		ClearWorkAreaLGVDone := TRUE;
		LGVAccessOK := FALSE;
		LGVCase := LGVCase + 1;	
		TFTimerSet(ADR(TimerOkBarriereSicurezze),5000, TRUE);	
		FOR iPost:=1 TO MAXAREAPRESENT DO
			IF LGV_Stato_Operazione^[k] = LGV_DEPOSITO_EFFETTUATO THEN  
				LGV_Stato_Operazione^[k] := LGV_OPERAZIONE_VERIFICATA;
				IF PH_WorkArea[k] THEN	//Se la fatocellula è ON
					IF TFMachinePalletizerMain.TEST_ENABLE THEN//Se sono in simulazione setto a TRUE la fotocellula virtuale
						I_PHPresenzaPalletVirtuale[k] := TRUE;
					ELSE
						//IF WorkArea^[k].Typology = TYPOLOGY_STACK OR WorkArea^[k].Typology = TYPOLOGY_LAYER THEN
						//	TFClearWorkAreaStack(WorkArea,WorkAreaState,k);
						//END_IF	
					END_IF
				ELSE 					//Se la fotocellula è OFF
					IF TFMachinePalletizerMain.TEST_ENABLE THEN//Se sono in simulazione setto a TRUE la fotocellula virtuale
						I_PHPresenzaPalletVirtuale[k] := TRUE;
					ELSE
						//IF WorkArea^[k].Typology = TYPOLOGY_STACK OR WorkArea^[k].Typology = TYPOLOGY_LAYER THEN
						//	TFClearWorkAreaStack(WorkArea,WorkAreaState,k);
						//END_IF	
						LGVErrorCode := ErrMACHINEPALLETIZER_PHOFFDOPODEPOSITO;
						LGVCase := 0;
					END_IF
				END_IF
			ELSIF LGV_Stato_Operazione^[k] = LGV_PRELIEVO_EFFETTUATO AND PH_WorkArea[k] THEN  
				LGV_Stato_Operazione^[k] := LGV_OPERAZIONE_VERIFICATA;
				IF NOT PH_WorkArea[k] THEN //Se la fotocellula è OFF
					IF TFMachinePalletizerMain.TEST_ENABLE THEN//Se sono in simulazione setto a FALSE la fotocellula virtuale
						I_PHPresenzaPalletVirtuale[k] := FALSE;
						TFClearWorkArea(WorkArea,WorkAreaState,k);
					ELSE
						TFClearWorkArea(WorkArea,WorkAreaState,k);
					END_IF
				ELSE					//Se la fotocellula è ON
					IF TFMachinePalletizerMain.TEST_ENABLE THEN//Se sono in simulazione setto a FALSE la fotocellula virtuale
						I_PHPresenzaPalletVirtuale[k] := FALSE;
						TFClearWorkArea(WorkArea,WorkAreaState,k);
					ELSE
						TFClearWorkArea(WorkArea,WorkAreaState,k);
					END_IF
					LGVErrorCode := ErrMACHINEPALLETIZER_PHONDOPOPRELIEVO;
					LGVCase := 0;
				END_IF
			ELSIF LGV_Stato_Operazione^[k] = LGV_OPERAZIONE_VERIFICATA THEN
				LGVErrorCode := ErrMACHINEPALLETIZER_MANCATOAGGIORNAMENTOSTATO;		
				LGVCase := 0;	
			END_IF
		END_FOR
			
	(* Case 7 - Power ON *)
	7:	
		IF BarriereSicurezzaEsterneOK THEN
			TFParametersArrayClear(ADR(ParametersArray));
			ParametersArray.Parameters[0] := '1';
			TFCommandSend(CmdPOWER,ParametersArray,MachineCmd^);
			LGV_ResetSW_RicIng := TRUE;
			LGVCase := LGVCase + 1;	
		ELSIF TFTimerDone(ADR(TimeoutControlloBarriereSicurezza)) THEN
			LGVErrorCode := ErrMACHINEPALLETIZER_BARRIEREOCCUPATE_LGVREQ_OFF;
			LGVCase := 0;
		END_IF	
			
	(* Case 8 - Power On OK *)
	8:	IF TFStateCodeGet(MachineState^) = StatePOWER_END OR
			TFIsModuleError(MachineError^) THEN
			LGV_ResetSW_RicIng := FALSE;
			LGVCase := LGVCase + 1;	
		END_IF
		
	(* Case 9 - Cmd DO *)
	9:	
		IF MachineWasRunning AND
			MachineMode^.Auto AND
			NOT MachineMode^.StopRequest AND
			NOT MachineMode^.RapidStopRequest AND NOT GateAccessActive THEN
			(*AND (SecurityGateStatus OR NOT ControlGateSecurity^*) 
			TFParametersArrayClear(ADR(ParametersArray));
			TFCommandSend(CmdDO,ParametersArray,MachineCmd^);
		END_IF
		LGVCase := 0;
	
	ELSE
		LGVAccessERROR := TRUE;
		LGVCase := 0;
	
END_CASE

(* Clocks *)
IF TFTimerDone(ADR(Timer100)) THEN
	TFTimerSet(ADR(Timer100),100,TRUE);
	Clock100 := NOT Clock100;
END_IF
IF TFTimerDone(ADR(Timer200)) THEN
	TFTimerSet(ADR(Timer200),200,TRUE);
	Clock200 := NOT Clock200;
END_IF
IF TFTimerDone(ADR(Timer1000)) THEN
	TFTimerSet(ADR(Timer1000),1000,TRUE);
	Clock1000 := NOT Clock1000;
END_IF

(* Se ho un errore durante la richiesta di ingresso, resetto esternamente gli HandShake *)
IF LGVErrorCode <> 0 THEN
	LGVResetHSKSUPNAV := TRUE;
END_IF


(* Access Lamp *)
LGVAccessLamp := ((LGVAccessOK AND Clock200) OR
				(LampadaIngressoInCorso AND Clock1000))AND
				NOT LGVAccessERROR OR (LGVAccessERROR AND Clock100);

END_FUNCTION_BLOCK

// ---- POUs/TFMachines/Utility/TFWorkflowsCheckState.TcPOU
FUNCTION TFWorkflowsCheckState : BOOL
VAR_INPUT
	WorkFlow : POINTER TO ARRAY[0..MAXWORKFLOW] OF WorkFlow;
	State : UINT; // stato da verificare
END_VAR
VAR
	i: UINT;
END_VAR
//Funzione che restituisce TRUE se tutti i WORFLOW sono nello stato richiesto

FOR i:=0 TO MAXWORKFLOW DO
	IF WorkFlow^[i].State <> State THEN
		RETURN;
	END_IF
END_FOR
TFWorkflowsCheckState := TRUE;

END_FUNCTION

// ---- POUs/TFModules/DataBase/TFSPRicavaDatiDaBarcodeUDC.TcPOU
FUNCTION_BLOCK TFSPRicavaDatiDaBarcodeUDC
VAR_INPUT
	BarcodeUDC 	: STRING;//Barcode in ingresso
	IDUDC 		: UDINT;//ID univoco che la macchina genera per ogni elemento depositato
	StartRead 	: BOOL;//Start lettura dati
	DBID		: UDINT;//ID del database, da ricavare dal configuratore
	AbilitaSTHere : BOOL;
	ResetError : bool;
END_VAR
VAR_OUTPUT
	DataFromDB 	: Record_From_DB; //Dati ricavati dal DB
	RecordID    : DINT; //se <> da 0 significa che l'elemento può entrare e rappresenta l'ordine di lavoro
	State 		: ARRAY [1..2] OF StoredProcedureState;
END_VAR
VAR
	nState: BYTE;
	arrParaList1: ARRAY [0..0] OF ST_DBParameter;
	arrParaList2: ARRAY [0..6] OF ST_DBParameter;
	SP_TryUdcCheckIn : FB_DBStoredProceduresRecordArray;
	SP_TryQtyCheckIn : FB_DBStoredProceduresRecordArray;

	bBusy: BOOL;
	bErr: BOOL;
	nErrid: UDINT;

	StateSP1 		: StoredProcedureState;
	StateSP2 		: StoredProcedureState;

	CalibroLocal : STRING;

END_VAR

CASE nState OF
	(*Idle*)
	0:
		IF StartRead THEN
			nState := 1;
			State[1].ReadRun := TRUE;
			DataFromDB.ArticleCode 	:= '';
			DataFromDB.Caliber		:= '';
			DataFromDB.Choice		:= '';
			DataFromDB.Length_mm	:= 0;
			DataFromDB.Quantity		:= 0;
			DataFromDB.Thickness_mm	:= 0;
			DataFromDB.Tone			:= '';
			DataFromDB.Udc			:= '';
			DataFromDB.Width_mm		:= 0;
		END_IF
	(* Case 1 : Init Dei parametri per esecuzione SP *)
	1:
		arrParaList1[0].sParameterName 		:= '@Udc';
		arrParaList1[0].eParameterDataType 	:= eDBColumn_NVarChar;
		arrParaList1[0].eParameterType 		:= eDBParameter_Input;
		arrParaList1[0].cbParameterValue 	:= SIZEOF(BarcodeUDC);
		arrParaList1[0].pParameterValue 		:= ADR(BarcodeUDC);
		SP_TryUdcCheckIn.bExecute := TRUE;
		
		(*SP_TryUdcCheckIn(
				sNetID	:= ,
				hDBID	:= DBID,
				sProcedureName	:= 'TryUdcCheckIn',
				cbParameterList	:= SIZEOF(arrParaList1),
				pParameterList	:= ADR(arrParaList1),
				nStartIndex		:= 0,
				nRecordCount	:= 1,
				cbRecordArraySize	:= SIZEOF(DataFromDB),
				pDestAddr			:= ADR(DataFromDB),
				//bExecute			:= TRUE,
				tTimeout			:= T#50S,
				bBusy				=> bBusy,
				bError				=> State[1].Error,
				nErrID				=> State[1].ErrorID,
				sSQLState			=> State[1].Sqlstate,
				nRecords			=> State[1].NumeroRecordLetti);	*)
		//IF NOT SP_TryUdcCheckIn.bBusy THEN
			nState := 2;
		//	SP_TryUdcCheckIn.bExecute := FALSE;
		//END_IF

	(*Start stored procedure "TryUdcCheckIn"*)
	2:
		IF NOT SP_TryUdcCheckIn.bBusy THEN
			SP_TryUdcCheckIn.bExecute := FALSE;
			IF AbilitaSTHere THEN
				nState := 10;
				RecordID := 0;
			ELSE
				nState := 12;
				State[2].ReadRun 	:= FALSE;
				State[2].ReadDone 	:= TRUE;
			END_IF
			State[1].ReadRun 	:= FALSE;
			State[1].ReadDone 	:= TRUE;
		END_IF
	
	10:
		//Parametro UDC generato dalla linea di ingresso
		arrParaList2[0].sParameterName 		:= '@IdEnteringUnit';
		arrParaList2[0].eParameterDataType 	:= eDBColumn_BigInt;
		arrParaList2[0].eParameterType 		:= eDBParameter_Input;
		arrParaList2[0].cbParameterValue 	:= SIZEOF(IDUDC);
		arrParaList2[0].pParameterValue 		:= ADR(IDUDC);

		//Parametro BARCODE
		arrParaList2[1].sParameterName 		:= '@UDC';
		arrParaList2[1].eParameterDataType 	:= eDBColumn_NVarChar;
		arrParaList2[1].eParameterType 		:= eDBParameter_Input;
		arrParaList2[1].cbParameterValue 	:= SIZEOF(BarcodeUDC);
		arrParaList2[1].pParameterValue 	:= ADR(BarcodeUDC);
		
		//Parametro Articolo
		arrParaList2[2].sParameterName 		:= '@Articolo';
		arrParaList2[2].eParameterDataType 	:= eDBColumn_NVarChar;
		arrParaList2[2].eParameterType 		:= eDBParameter_Input;
		arrParaList2[2].cbParameterValue 	:= SIZEOF(DataFromDB.ArticleCode);
		arrParaList2[2].pParameterValue 		:= ADR(DataFromDB.ArticleCode);
		//Parametro Scelta
		arrParaList2[3].sParameterName 		:= '@Scelta';
		arrParaList2[3].eParameterDataType 	:= eDBColumn_NVarChar;
		arrParaList2[3].eParameterType 		:= eDBParameter_Input;
		arrParaList2[3].cbParameterValue 	:= SIZEOF(DataFromDB.Choice);
		arrParaList2[3].pParameterValue 		:= ADR(DataFromDB.Choice);

		//Parametro tono
		arrParaList2[4].sParameterName 		:= '@Tono';
		arrParaList2[4].eParameterDataType 	:= eDBColumn_NVarChar;
		arrParaList2[4].eParameterType 		:= eDBParameter_Input;
		arrParaList2[4].cbParameterValue 	:= SIZEOF(DataFromDB.Tone);
		arrParaList2[4].pParameterValue 		:= ADR(DataFromDB.Tone);

		//Parametro Calibro
		arrParaList2[5].sParameterName 		:= '@Calibro';
		arrParaList2[5].eParameterDataType 	:= eDBColumn_NVarChar;
		arrParaList2[5].eParameterType 		:= eDBParameter_Input;

		arrParaList2[5].cbParameterValue 	:= SIZEOF(DataFromDB.Caliber);
		arrParaList2[5].pParameterValue 		:= ADR(DataFromDB.Caliber);
		//Parametro Quantità
		arrParaList2[6].sParameterName 		:= '@Quantity';
		arrParaList2[6].eParameterDataType 	:= eDBColumn_Float;
		arrParaList2[6].eParameterType 		:= eDBParameter_Input;
		arrParaList2[6].cbParameterValue 	:= SIZEOF(DataFromDB.Quantity);
		arrParaList2[6].pParameterValue 	:= ADR(DataFromDB.Quantity);
		//Reset variabile risultante
		//RecordID := 0;
		//Lancio Comando
		SP_TryQtyCheckIn.bExecute := TRUE;

		(*SP_TryQtyCheckIn(
				sNetID	:= ,
				hDBID	:= DBID,
				sProcedureName	:= 'TryQtyCheckIn',
				cbParameterList	:= SIZEOF(arrParaList2),
				pParameterList	:= ADR(arrParaList2),
				nStartIndex		:= 0,
				nRecordCount	:= 1,
				cbRecordArraySize	:= SIZEOF(RecordID),
				pDestAddr			:= ADR(RecordID),
				//bExecute			:= TRUE,
				tTimeout			:= T#50S,
				bBusy				=> bBusy,
				bError				=> State[2].Error,
				nErrID				=> State[2].ErrorID,
				sSQLState			=> State[2].Sqlstate,
				nRecords			=> State[2].NumeroRecordLetti);*)
		
		State[2].ReadRun 	:= TRUE;
		State[2].ReadDone 	:= FALSE;

		//IF NOT SP_TryQtyCheckIn.bBusy THEN
		//	SP_TryQtyCheckIn.bExecute := FALSE;
			nState := 11;
		//END_IF

	(*Start stored procedure "TryUdcCheckIn"*)
	11:
		IF NOT SP_TryQtyCheckIn.bBusy THEN
			SP_TryQtyCheckIn.bExecute := FALSE;
			nState := 12;//3;
			State[2].ReadRun 	:= FALSE;
			State[2].ReadDone 	:= TRUE;
		END_IF

	(* Attesa che il comando dall'esterno venga azzerato *)	
	12:
		IF NOT StartRead OR ResetError THEN 
			nState := 0;
			State[1].ReadRun 	:= FALSE;
			State[2].ReadRun 	:= FALSE;
			State[1].ReadDone 	:= FALSE;
			State[2].ReadDone 	:= FALSE;
			SP_TryUdcCheckIn.bExecute := FALSE;
			SP_TryQtyCheckIn.bExecute := FALSE;
			
		END_IF	
		
END_CASE

//Lancio SP
(*
IF ResetError THEN
	IF SP_TryUdcCheckIn.bError AND NOT SP_TryUdcCheckIn.bBusy THEN
		SP_TryUdcCheckIn.bExecute := FALSE;
		//SP_TryUdcCheckIn(bExecute := FALSE);
	END_IF
	IF  SP_TryQtyCheckIn.bError AND NOT SP_TryUdcCheckIn.bBusy THEN 
		SP_TryQtyCheckIn.bExecute := FALSE;
		//SP_TryQtyCheckIn(bExecute := FALSE);
	END_IF
	ResetError := FALSE;
END_IF
*)

SP_TryUdcCheckIn(
				sNetID	:= ,
				hDBID	:= DBID,
				sProcedureName	:= 'TryUdcCheckIn',
				cbParameterList	:= SIZEOF(arrParaList1),
				pParameterList	:= ADR(arrParaList1),
				nStartIndex		:= 0,
				nRecordCount	:= 1,
				cbRecordArraySize	:= SIZEOF(DataFromDB),
				pDestAddr			:= ADR(DataFromDB),
				//bExecute			:= TRUE,
				tTimeout			:= T#50S,
				bBusy				=> bBusy,
				bError				=> State[1].Error,
				nErrID				=> State[1].ErrorID,
				sSQLState			=> State[1].Sqlstate,
				nRecords			=> State[1].NumeroRecordLetti);

//Lancio SP
SP_TryQtyCheckIn(
				sNetID	:= ,
				hDBID	:= DBID,
				sProcedureName	:= 'TryQtyCheckIn',
				cbParameterList	:= SIZEOF(arrParaList2),
				pParameterList	:= ADR(arrParaList2),
				nStartIndex		:= 0,
				nRecordCount	:= 1,
				cbRecordArraySize	:= SIZEOF(RecordID),
				pDestAddr			:= ADR(RecordID),
				//bExecute			:= TRUE,
				tTimeout			:= T#50S,
				bBusy				=> bBusy,
				bError				=> State[2].Error,
				nErrID				=> State[2].ErrorID,
				sSQLState			=> State[2].Sqlstate,
				nRecords			=> State[2].NumeroRecordLetti);

//reset errori SP				
IF ResetError THEN
	IF State[1].Error THEN
		State[1].Error := FALSE;
	END_IF
	IF State[2].Error THEN 
		State[2].Error := FALSE;
	END_IF
	ResetError := FALSE;
END_IF

END_FUNCTION_BLOCK

// ---- POUs/TFModules/DataBase/TFSPRichiestaIngressoMateriale.TcPOU
FUNCTION_BLOCK TFSPRichiestaIngressoMateriale
VAR_INPUT
	BarcodeUDC 	: STRING;//Barcode in ingresso
	StartRead 	: BOOL;//Start lettura dati
	DBID		: UDINT;//ID del database, da ricavare dal configuratore
END_VAR
VAR_OUTPUT
	DataFromDB 	: Record_From_DB; //Dati ricavati dal DB
	State 		: StoredProcedureState;
END_VAR
VAR
	nState: BYTE;
	arrParaList: ARRAY [0..0] OF ST_DBParameter;
	SP_RecordArray : FB_DBStoredProceduresRecordArray;
	bBusy: BOOL;
	bErr: BOOL;
	nErrid: UDINT;
	DataFromDB1 	: Record_From_DB; //Dati ricavati dal DB
END_VAR

CASE nState OF
	(*Idle*)
	0:
		IF StartRead THEN
			nState := 1;
			State.ReadRun := TRUE;
		END_IF
	(* Case 1 : Init Dei parametri per esecuzione SP *)
	1:
		arrParaList[0].sParameterName 		:= '@Udc';
		arrParaList[0].eParameterDataType 	:= eDBColumn_NVarChar;
		arrParaList[0].eParameterType 		:= eDBParameter_Input;
		arrParaList[0].cbParameterValue 	:= SIZEOF(BarcodeUDC);
		arrParaList[0].pParameterValue 		:= ADR(BarcodeUDC);
	
		DataFromDB.ArticleCode 	:= '';
		DataFromDB.Caliber		:= '';
		DataFromDB.Choice		:= '';
		DataFromDB.Length_mm	:= 0;
		DataFromDB.Quantity		:= 0;
		DataFromDB.Thickness_mm	:= 0;
		DataFromDB.Tone			:= '';
		DataFromDB.Udc			:= '';
		DataFromDB.Width_mm		:= 0;

		SP_RecordArray.bExecute := TRUE;
		
		nState := 2;

	(*Start stored procedure "TryUdcCheckIn"*)
	2:
		
		
		IF NOT SP_RecordArray.bBusy THEN
			SP_RecordArray.bExecute := FALSE;
			nState := 3;
			State.ReadRun 	:= FALSE;
			State.ReadDone 	:= TRUE;
		END_IF
	
	(* Attesa che il comando dall'esterno venga azzerato *)	
	3:
		IF NOT StartRead THEN 
			nState := 0;
			State.ReadRun 	:= FALSE;
			State.ReadDone 	:= FALSE;
		END_IF	
		
END_CASE

//Lancio FB
SP_RecordArray(
				sNetID	:= ,
				hDBID	:= DBID,
				sProcedureName	:= 'TryUdcCheckIn',
				cbParameterList	:= SIZEOF(arrParaList),
				pParameterList	:= ADR(arrParaList),
				nStartIndex		:= 0,
				nRecordCount	:= 1,
				cbRecordArraySize	:= SIZEOF(DataFromDB1),
				pDestAddr			:= ADR(DataFromDB1),
				//bExecute			:= TRUE,
				tTimeout			:= T#50S,
				bBusy				=> bBusy,
				bError				=> State.Error,
				nErrID				=> State.ErrorID,
				sSQLState			=> State.Sqlstate,
				nRecords			=> State.NumeroRecordLetti);

END_FUNCTION_BLOCK

// ---- POUs/TFModules/DataBase/TFVerificaLetturaBarcodeConDatiDB.TcPOU
FUNCTION_BLOCK TFVerificaLetturaBarcodeConDatiDB //FB che verifica se i dati letti del barcode sono validi per il database
VAR_INPUT
	VerificaDati 	: BOOL;	//Bit di start
	BarcodeUDC 		: STRING;//Barcode elemento
	IDUDC 			: UDINT;//ID elemento
	AbilitaSTHere 	: BOOL;
END_VAR
VAR
	DataElementNull : TFMachinePalletizer_DataElement;
	DimElementNull	: TFDimensionElement; 
	RicavaDatiDaBarcodeUDC : TFSPRicavaDatiDaBarcodeUDC;
	FirstCycleDone : bool;
END_VAR
VAR_OUTPUT
	DatoValido 			: BOOL; //Dati ok
	VerificaDatiDone 	: BOOL; //Verifica completata
	DataElement 		: TFMachinePalletizer_DataElement;//dati elemento
	DimElement 			: TFDimensionElement; //Dimensioni Pezzi
	RequetsIDValido		: BOOL;//se TRUE allora il materiale puù entrare
	Error : BOOL;
END_VAR


IF VerificaDati AND BarcodeUDC <> '0' AND BarcodeUDC <> '' AND NOT (RicavaDatiDaBarcodeUDC.State[1].Error OR RicavaDatiDaBarcodeUDC.State[2].Error) THEN//Se ho il comando di verifica dei dati su DB
	Error 			:= FALSE;
	RicavaDatiDaBarcodeUDC.ResetError := FALSE;
	RequetsIDValido := FALSE;
	DataElement 	:= DataElementNull;
	DimElement 		:= DimElementNull;
	AbilitaSTHere 	:= TRUE;	

	(* Eseguo Stored Procedure per acquisire i dati dell'articolo all'interno dell'UDC avente il codice in ingresso del BARCODE *)
	RicavaDatiDaBarcodeUDC.BarcodeUDC 	:= BarcodeUDC; 	//BARCODE letto sull'elemento
	RicavaDatiDaBarcodeUDC.DBID 		:= 1;			//Numero del DB configurato
	RicavaDatiDaBarcodeUDC.IDUDC 		:= IDUDC;		//ID dell'elemento
	RicavaDatiDaBarcodeUDC.StartRead 	:= TRUE;		//Start comando lettura
	RicavaDatiDaBarcodeUDC.AbilitaSTHere := AbilitaSTHere;	

	IF (RicavaDatiDaBarcodeUDC.State[1].ReadDone AND NOT RicavaDatiDaBarcodeUDC.State[1].Error) THEN
		//Dati elemento
		DataElement.Tono 	:= RicavaDatiDaBarcodeUDC.DataFromDB.Tone;
		DataElement.Scelta 	:= RicavaDatiDaBarcodeUDC.DataFromDB.Choice;
		DataElement.Calibro := RicavaDatiDaBarcodeUDC.DataFromDB.Caliber;
		DataElement.Codice  := RicavaDatiDaBarcodeUDC.DataFromDB.ArticleCode;
		DataElement.Quantity := LREAL_TO_UINT(RicavaDatiDaBarcodeUDC.DataFromDB.Quantity);
		DataElement.ArticleDescription  := RicavaDatiDaBarcodeUDC.DataFromDB.ArticleDescription;
		
		//Dimensioni elemento
		DimElement.ZDim		:= DINT_TO_REAL(RicavaDatiDaBarcodeUDC.DataFromDB.Thickness_mm);
		IF RicavaDatiDaBarcodeUDC.DataFromDB.Length_mm > RicavaDatiDaBarcodeUDC.DataFromDB.Width_mm THEN
			DimElement.XDim		:= DINT_TO_REAL(RicavaDatiDaBarcodeUDC.DataFromDB.Length_mm);
			DimElement.YDim		:= DINT_TO_REAL(RicavaDatiDaBarcodeUDC.DataFromDB.Width_mm);
		ELSE
			DimElement.XDim		:= DINT_TO_REAL(RicavaDatiDaBarcodeUDC.DataFromDB.Width_mm);
			DimElement.YDim		:= DINT_TO_REAL(RicavaDatiDaBarcodeUDC.DataFromDB.Length_mm);
		END_IF

		//Validità dati
		DatoValido 			:= NOT RicavaDatiDaBarcodeUDC.State[1].Error AND DataElement.Codice <> '0' AND DataElement.Codice <> '';
		 
		IF ((RicavaDatiDaBarcodeUDC.State[2].ReadDone AND NOT RicavaDatiDaBarcodeUDC.State[2].Error) OR NOT AbilitaSTHere) THEN//Se lettura da DB terminata	
			//Valore Record ID che se <> da 0 vuol dire che il materiale puù entrare
			IF NOT RicavaDatiDaBarcodeUDC.State[2].Error THEN
				DataElement.WorkingID 	:= DINT_TO_STRING(RicavaDatiDaBarcodeUDC.RecordID);
				RequetsIDValido 		:= DataElement.WorkingID <> '0';//indico che l'elemento può entrare
				IF NOT RequetsIDValido THEN
					DataElement.WorkingID := '0';
				END_IF
			ELSE
				DataElement.WorkingID 	:= '';
			END_IF
		END_IF
		RicavaDatiDaBarcodeUDC.StartRead := FALSE;//Stoppo la lettura
		VerificaDatiDone 	:= TRUE;
	ELSIF FirstCycleDone AND RicavaDatiDaBarcodeUDC.State[1].Error OR RicavaDatiDaBarcodeUDC.State[2].Error THEN
		Error 				:= TRUE;
		VerificaDatiDone 	:= TRUE;
		RicavaDatiDaBarcodeUDC.StartRead := FALSE;//Stoppo la lettura
	END_IF
	FirstCycleDone := TRUE;
	
ELSIF VerificaDatiDone AND NOT VerificaDati THEN //Attendo che dall'esterno venga terminata la richiesta di lettura dal DB
	DatoValido 			:= FALSE;
	VerificaDatiDone 	:= FALSE;
	FirstCycleDone 		:= FALSE;
ELSIF RicavaDatiDaBarcodeUDC.State[1].Error OR RicavaDatiDaBarcodeUDC.State[2].Error THEN
	DatoValido 	:= FALSE;
	RicavaDatiDaBarcodeUDC.ResetError := TRUE;
	Error 				:= TRUE;
END_IF

//Esguo FB per ricerca dati da DB
RicavaDatiDaBarcodeUDC();

END_FUNCTION_BLOCK

// ---- POUs/TFModules/Misurazione Ingresso/TFGestioneFTC_Misura.TcPOU
FUNCTION_BLOCK TFGestioneFTC_Misura
VAR_INPUT
	EseguiMisura 	: BOOL; //Start esecuzione misura
	IN 				: TFGestioneFTC_Misura_IN; //Struttura Ingressi
	PosizioneAsse 	: LREAL;	//Posizione dell'asse
	AsseInMovimento : BOOL; //Indica se l'asse è in movimento o meno
	SpazioFiltro 	: REAL := 50; //Spazio utilizzato per filtrare le FTC
END_VAR
VAR_OUTPUT
	
	OUT 				: TFGestioneFTC_Misura_OUT;
END_VAR
VAR
	FiltroFTC1 : Signal_SpaceFilter;
	FiltroFTC2 : Signal_SpaceFilter;
	FiltroFTC3 : Signal_SpaceFilter;
	FiltroFTC4 : Signal_SpaceFilter;
	
	StartLettura 	: BOOL;
	PosizioneTesta 	: REAL;
	PosizioneCoda 	: REAL;
	
	UltimaLunghezza : REAL := 0; //Appoggio x debug
	FTC_PallettoneIntercettata : BOOL;
END_VAR

FiltroFTC1(Sensor:=IN.FTC_ZoccoloBasso,
			ActualPosition:=PosizioneAsse,
			SpaceFilter:=SpazioFiltro,
			AxisMoving:=AsseInMovimento,
			EnableDirectStatusAxStop:=TRUE,
			SensorOUT=>OUT.FTC_ZoccoloBassoFiltrata);
FiltroFTC2(Sensor:=IN.FTC_Pallettone,
			ActualPosition:=PosizioneAsse,
			SpaceFilter:=SpazioFiltro,
			AxisMoving:=AsseInMovimento,
			EnableDirectStatusAxStop:=TRUE,
			SensorOUT=>OUT.FTC_PallettoneFiltrata);
FiltroFTC3(Sensor:=IN.FTC_CavallinaBassa,
			ActualPosition:=PosizioneAsse,
			SpaceFilter:=SpazioFiltro,
			AxisMoving:=AsseInMovimento,
			EnableDirectStatusAxStop:=TRUE,
			SensorOUT=>OUT.FTC_CavallinaBassaFiltrata);
FiltroFTC4(Sensor:=IN.FTC_CavallinaAlta,
			ActualPosition:=PosizioneAsse,
			SpaceFilter:=SpazioFiltro,
			AxisMoving:=AsseInMovimento,
			EnableDirectStatusAxStop:=TRUE,
			SensorOUT=>OUT.FTC_CavallinaAltaFiltrata);

IF EseguiMisura THEN
	IF OUT.FTC_ZoccoloBassoFiltrata THEN
		//Memorizzo la quota della testa dell'elemento
		IF NOT StartLettura THEN 
			Out.Supporto := SupportoVuoto;//Sbianco la memoria dell'ultima lettura
			UltimaLunghezza := 0;
			OUT.MisuraInCorso := TRUE;  
			PosizioneTesta := PosizioneAsse;
			StartLettura := TRUE;
		END_IF	
	
		IF OUT.FTC_PallettoneFiltrata OR WEINTEK_TRANSPORT.AbilitaIngressoPalletSingolo THEN //Se vedo questa FTC sicuramente non è una cassa
			IF NOT WEINTEK_TRANSPORT.AbilitaIngressoPalletSingolo THEN
				OUT.Supporto.Tipologia := PALLET_ACCOPPIATI;//Dichiaro la tipologia di supporto
			ELSE
				OUT.Supporto.Tipologia := PALLET_STANDARD;//Dichiaro la tipologia di supporto
			END_IF
			OUT.Supporto.ZDim := 1000;//800;
			OUT.Supporto.HMAX := 1000;//800;
			FTC_PallettoneIntercettata := TRUE;
			IF OUT.FTC_CavallinaBassaFiltrata THEN //Se vedo questa FTC si tratta di una cavallina Bassa
				OUT.Supporto.Tipologia := CAVALLETTO;//Dichiaro la tipologia di supporto
				OUT.Supporto.ZDim := 350;
				OUT.Supporto.HMAX := 1600;
			END_IF
			IF OUT.FTC_CavallinaAltaFiltrata THEN //Se vedo questa FTC si tratta di cavallina ALTA
				OUT.Supporto.Tipologia := CAVALLETTO;//Dichiaro la tipologia di supporto
				OUT.Supporto.ZDim := 350;
				OUT.Supporto.HMAX := 2000;
			END_IF
		ELSIF NOT OUT.FTC_PallettoneFiltrata AND NOT FTC_PallettoneIntercettata THEN //Se non vedo questa FTC si tratta di una cassa
			OUT.Supporto.Tipologia := CASSA_STANDARD;//Dichiaro la tipologia di supporto
			OUT.Supporto.ZDim := 200;
			OUT.Supporto.HMAX := 420;
		END_IF
	
	ELSIF NOT OUT.FTC_ZoccoloBassoFiltrata AND StartLettura THEN
		Out.MisuraDone := TRUE;
		OUT.MisuraInCorso := TRUE;  
		PosizioneCoda := PosizioneAsse;
		Out.LunghezzaMisurata := PosizioneCoda - PosizioneTesta;
		Out.Supporto.XDim := Out.LunghezzaMisurata;
		UltimaLunghezza := Out.LunghezzaMisurata;
		FTC_PallettoneIntercettata := FALSE;
	END_IF
	//Cambio tipologia nel caso di pallet >= 1400
	IF Out.Supporto.XDim >= 1400 AND OUT.Supporto.Tipologia = PALLET_ACCOPPIATI THEN
		OUT.Supporto.Tipologia := PALLET_STANDARD;
	END_IF
ELSE
	Out.MisuraDone 		:= FALSE;
	OUT.MisuraInCorso 	:= FALSE;
	StartLettura 		:= FALSE;
	
END_IF

END_FUNCTION_BLOCK

// ---- POUs/TFModules/Moduli TF/TFModulePalletizer_Pinza_mag.TcPOU
FUNCTION_BLOCK TFModulePalletizer_Pinza_mag
VAR_INPUT
	Cmd 	: CommandBuffer;
	Cfg 	: Config;
	IN 		: TFMchinePalletizer_PinzaVentose_IN;
	IN_Ax 	: Module_Palletizer_Ax_IN;
	
	AspirazioneDX1 : POINTER TO TF_VacumOVEM;
	AspirazioneSX1 : POINTER TO TF_VacumOVEM;
	AspirazioneDX2 : POINTER TO TF_VacumOVEM;
	AspirazioneSX2 : POINTER TO TF_VacumOVEM;

	CilindroSbloccoRotazione 	: POINTER TO SC_Cylinder;
	CilindroSbloccoBascolante 	: POINTER TO SC_Cylinder;
	CilindroApertura 			: POINTER TO DC_Cylinder;
	
	ModuleJ : POINTER TO TFModulePalletizer_Ax;
	ModuleK : POINTER TO TFModulePalletizer_Ax;

	ManCmd 				: POINTER TO TFMachinePalletizer_PinzaVentoseManCmd;
	ElementoInPrelievo 	: TFMachinePalletizer_PlaceElement;
	DataElement			: TFMachinePalletizer_DataElement; (* Struttura dati che la macchina acquisisce/trasferisce in fase di pallettizzazione/depallettizazione *)
	PrelievoSuMagazino : BOOL;//indica che il prelievo è su cavallina

	Mission : POINTER TO TFMachinePalletizer_Mission;
	AbilitazioneSbloccoRotazione 	: BOOL;//Abilitazione sblocco rotazione pinza
	AbilitazioneSbloccoBascolante 	: BOOL;//Abilitazione sblocco bascolante pinza	
	IN_SimulazioneSenzaHW : BOOL;
	AbilitaAperturaAutomaticaPinza : BOOL;//Abilitazione apertura automatica pinza
END_VAR
VAR_OUTPUT
	CmdExe 		: CommandExe;
	CmdExd 		: CommandExe;
	CmdNext 	: Command;
	CmdLog 		: CommandLog;
	ProgramLog 	: ProgrammaLog; 
	State 		: State;
	StateLog 	: StateLog;
	Error 		: Error;
	ErrorLog 	: ErrorLog;
	Warning 	: Warning;
	WarningLog	: WarningLog;
	OUT 		: TFMachinePalletizer_PinzaVentose_OUT;
	StatoPinza 	: TFMachinePalletizer_PinzaState;

END_VAR
VAR
	Power 	: UINT;
	Init 	: BOOL;
	Timer 	: REAL;
	Timeout : REAL;
	TimerAspirazione 	: REAL;
	ParametersArray 	: ParametersArray;
	MAN_Actuator 		: UINT;
	MAN_Cmd 			: UINT;

	DistanzaFTC_J0 		: REAL;
	DistanzaFTC_J180 	: REAL;
	DistanzaFTC_K0 		: REAL;
	DistanzaFTC_K180 	: REAL;

	TimerPresaPiastrella : REAL;		
	DisattivazioneTotaleAspirazioni : bool;
	ByPassAttesaDistacco : BOOL;

	DistanzaJForzata : REAL;
	DistanzaKForzata : REAL;

END_VAR

IF NOT Init THEN
	TFCommandBufferClear(ADR(Cmd));
	TFCommandClear(ADR(CmdNext));
	TFCommandExeClear(ADR(CmdExe));
	TFStateUpdate(ADR(State),StateNOP);
	TFErrorClear(ADR(Error));
	TFWarningClear(ADR(Warning));
	Init := TRUE;
END_IF

(* Generic Timer - Add here all your Timers *)
TFTimerCall(ADR(Timer),Cfg.TimeBase);
TFTimerCall(ADR(Timeout),Cfg.TimeBase);
TFTimerCall(ADR(TimerPresaPiastrella),Cfg.TimeBase);
TFTimerCall(ADR(TimerAspirazione),Cfg.TimeBase);
(* External To Buffered Command *)
TFCommandToNext(ADR(Cmd),ADR(CmdNext),ADR(CmdExe),ADR(Cfg),ADR(Error),ADR(ErrorLog),ADR(State));

(* Buffered To Exe Command *)
TFCommandToExecution(ADR(CmdNext),ADR(CmdExe),ADR(Error),ADR(ErrorLog),ADR(State),ADR(CmdLog));

(* Chiamata FB *)
AspirazioneDX1^();
AspirazioneSX1^();
AspirazioneDX2^();
AspirazioneSX2^();
CilindroSbloccoRotazione^();
CilindroSbloccoBascolante^();

DistanzaFTC_J0 		:= Keyence_LRTB2000C(IN.InKeyence_J0_Byte0,IN.InKeyence_J0_Byte1);
DistanzaFTC_J180	:= Keyence_LRTB2000C(IN.InKeyence_J180_Byte0,IN.InKeyence_J180_Byte1);
DistanzaFTC_K0 		:= Keyence_LRTB2000C(IN.InKeyence_K0_Byte0,IN.InKeyence_K0_Byte1);
DistanzaFTC_K180	:= Keyence_LRTB2000C(IN.InKeyence_K180_Byte0,IN.InKeyence_K180_Byte1);

OUT.DistanzaFTC_J0 		:= DistanzaFTC_J0; 		
OUT.DistanzaFTC_J180	:= DistanzaFTC_J180;	
OUT.DistanzaFTC_K0 		:= DistanzaFTC_K0; 		
OUT.DistanzaFTC_K180   	:= DistanzaFTC_K180; 

DistanzaJForzata:=0;
IF ABS(DistanzaFTC_J0-DistanzaFTC_J180) > 30 THEN
	DistanzaJForzata := MIN(DistanzaFTC_J0,DistanzaFTC_J180);
END_IF
DistanzaKForzata:=0;
IF ABS(DistanzaFTC_K0-DistanzaFTC_K180) > 30 THEN
	DistanzaKForzata := MIN(DistanzaFTC_K0,DistanzaFTC_K180);
END_IF
OUT.DistanzaMedia := (DistanzaFTC_J0 + 	
                 DistanzaFTC_J180 +
                 DistanzaFTC_K0 + 	
                 DistanzaFTC_K180)/4;
				 
IF DistanzaKForzata > 0 THEN
	OUT.DistanzaMedia := (DistanzaJForzata +
                 DistanzaFTC_K0 + 	
                 DistanzaFTC_K180)/3;
END_IF
IF DistanzaJForzata > 0 THEN
	OUT.DistanzaMedia := (DistanzaFTC_J0 + 	
                 DistanzaFTC_J180 +
                 DistanzaKForzata)/3;
END_IF
IF DistanzaKForzata > 0 AND DistanzaJForzata > 0 THEN
	OUT.DistanzaMedia := (DistanzaJForzata +
                 DistanzaKForzata)/2;
END_IF

(* Exe Command *)
CASE CmdExe.Code OF

	(* ******************************************************************************************************** *)
	(* Nop  *)
	(* ******************************************************************************************************** *)
	CmdNOP:	;			
	(* ******************************************************************************************************** *)
	(* Stop *)
	(* ******************************************************************************************************** *)
	CmdSTOP:
		CASE CmdExe.CmdCase OF
			
			(* Case 0 *)
			0: 	TFStateUpdate(ADR(State),StateSTOP_RUN);
				TFTimerSet(ADR(Timeout),500,TRUE);
				TFCommandCase(ADR(CmdExe),1,CommandCase_INC);

			(* Case 1 - Clear All Commands*)
			1:	
				TFCommandCase(ADR(CmdExe),100,CommandCase_JMP);
			(* Case 100 *)
			100:TFStateUpdate(ADR(State),StateSTOP_END);
				TFCommandExeClear(ADR(CmdExe));

			ELSE
				TFError(ErrNOCMDCASE,ErrNULL,ADR(CmdExe),ADR(State),ADR(Error),ADR(ErrorLog));
		END_CASE;
	
	(* ******************************************************************************************************** *)
	(* Error Reset *)
	(* ******************************************************************************************************** *)
	CmdRESET:
		CASE CmdExe.CmdCase OF

			(* Case 0 *)
			0: 	TFStateUpdate(ADR(State),StateRESET_RUN);
				TFTimerSet(ADR(Timeout),2000+100,TRUE);
				TFTimerSet(ADR(Timer),2000,TRUE);
				TFCommandCase(ADR(CmdExe),1,CommandCase_JMP);

			
			(* Case 1 - RESET COMANDI*)
			1: 
				TFClearAllCmdModulePinzaMagazzino(AspirazioneDX1,AspirazioneSX1,AspirazioneDX2,AspirazioneSX2,CilindroSbloccoRotazione,CilindroSbloccoBascolante);
				TFCommandCase(ADR(CmdExe),1,CommandCase_INC);
			
			(* Case 2 - Invio comando di reset *)
			2:
				AspirazioneDX1^.Command^.ErrorReset 				:= TRUE;	
				AspirazioneSX1^.Command^.ErrorReset 				:= TRUE;	
				AspirazioneDX2^.Command^.ErrorReset 				:= TRUE;	
				AspirazioneSX2^.Command^.ErrorReset 				:= TRUE;	
				CilindroSbloccoRotazione^.Command.ErrorReset 	:= TRUE;	
				CilindroSbloccoBascolante^.Command.ErrorReset 	:= TRUE;	
				TFCommandCase(ADR(CmdExe),1,CommandCase_INC);
			
			(* Case 3 - Invio comando di reset *)
			3:
				IF (AspirazioneDX1^.Status.ErrorResetDone AND AspirazioneDX2^.Status.ErrorResetDone AND
					AspirazioneSX1^.Status.ErrorResetDone AND AspirazioneSX2^.Status.ErrorResetDone AND
					CilindroSbloccoRotazione^.Status.ErrorResetDone AND CilindroSbloccoBascolante^.Status.ErrorResetDone) OR IN_SimulazioneSenzaHW THEN					
					TFClearAllCmdModulePinzaMagazzino(AspirazioneDX1,AspirazioneSX1,AspirazioneDX2,AspirazioneSX2,CilindroSbloccoRotazione,CilindroSbloccoBascolante);
					TFCommandCase(ADR(CmdExe),99,CommandCase_JMP);
				ELSIF TFTimerDone(ADR(Timer)) THEN
					TFClearAllCmdModulePinzaMagazzino(AspirazioneDX1,AspirazioneSX1,AspirazioneDX2,AspirazioneSX2,CilindroSbloccoRotazione,CilindroSbloccoBascolante);
					TFError(ErrTORESET,ErrNULL,ADR(CmdExe),ADR(State),ADR(Error),ADR(ErrorLog));
				END_IF

			(* Case 99 *)
			99:	TFErrorClear(ADR(Error));
				TFWarningClear(ADR(Warning));
				TFCommandCase(ADR(CmdExe),100,CommandCase_JMP);

			(* Case 100 *)
			100:TFStateUpdate(ADR(State),StateRESET_END);
				TFCommandExeClear(ADR(CmdExe));

			ELSE
				TFError(ErrNOCMDCASE,ErrNULL,ADR(CmdExe),ADR(State),ADR(Error),ADR(ErrorLog));
		END_CASE;

		(*IF AspirazioneDX^.Status.ErrorID <> ErrNULL THEN
			TFClearAllCmdModulePinza(AspirazioneDX,AspirazioneSX,CilindroApertura,CilindroSbloccoRotazione,AspirazioneFaldaDX,AspirazioneFaldaSX,CilindroTasteggio);
			TFError(ErrCYLINDER,AspirazioneDX^.Status.ErrorID,ADR(CmdExe),ADR(State),ADR(Error),ADR(ErrorLog));
		ELSIF AspirazioneSX^.Status.ErrorID <> ErrNULL THEN
			TFClearAllCmdModulePinza(AspirazioneDX,AspirazioneSX,CilindroApertura,CilindroSbloccoRotazione,AspirazioneFaldaDX,AspirazioneFaldaSX,CilindroTasteggio);
			TFError(ErrCYLINDER,AspirazioneSX^.Status.ErrorID,ADR(CmdExe),ADR(State),ADR(Error),ADR(ErrorLog));
		ELSIF CilindroApertura^.Status.ErrorID <> ErrNULL THEN
			TFClearAllCmdModulePinza(AspirazioneDX,AspirazioneSX,CilindroApertura,CilindroSbloccoRotazione,AspirazioneFaldaDX,AspirazioneFaldaSX,CilindroTasteggio);
			TFError(ErrCYLINDER,CilindroApertura^.Status.ErrorID,ADR(CmdExe),ADR(State),ADR(Error),ADR(ErrorLog));
		ELSIF CilindroSbloccoRotazione^.Status.ErrorID <> ErrNULL THEN
			TFClearAllCmdModulePinza(AspirazioneDX,AspirazioneSX,CilindroApertura,CilindroSbloccoRotazione,AspirazioneFaldaDX,AspirazioneFaldaSX,CilindroTasteggio);
			TFError(ErrCYLINDER,CilindroSbloccoRotazione^.Status.ErrorID,ADR(CmdExe),ADR(State),ADR(Error),ADR(ErrorLog));
		ELSIF AspirazioneFaldaDX^.Status.ErrorID <> ErrNULL THEN
			TFClearAllCmdModulePinza(AspirazioneDX,AspirazioneSX,CilindroApertura,CilindroSbloccoRotazione,AspirazioneFaldaDX,AspirazioneFaldaSX,CilindroTasteggio);
			TFError(ErrCYLINDER,AspirazioneFaldaDX^.Status.ErrorID,ADR(CmdExe),ADR(State),ADR(Error),ADR(ErrorLog));
		ELSIF AspirazioneFaldaSX^.Status.ErrorID <> ErrNULL THEN
			TFClearAllCmdModulePinza(AspirazioneDX,AspirazioneSX,CilindroApertura,CilindroSbloccoRotazione,AspirazioneFaldaDX,AspirazioneFaldaSX,CilindroTasteggio);
			TFError(ErrCYLINDER,AspirazioneFaldaSX^.Status.ErrorID,ADR(CmdExe),ADR(State),ADR(Error),ADR(ErrorLog));
		*)
		IF TFTimerDone(ADR(Timeout)) THEN
			TFClearAllCmdModulePinzaMagazzino(AspirazioneDX1,AspirazioneSX1,AspirazioneDX2,AspirazioneSX2,CilindroSbloccoRotazione,CilindroSbloccoBascolante);
			TFError(ErrCMDTIMEOUT,ErrNULL,ADR(CmdExe),ADR(State),ADR(Error),ADR(ErrorLog));
		END_IF
	
	(* ******************************************************************************************************** *)
	(* Power *)
	(* ******************************************************************************************************** *)
	CmdPOWER:
		CASE CmdExe.CmdCase OF
			
			(* Case 0 *)
			0: 	TFStateUpdate(ADR(State),StatePOWER_RUN);
				TFTimerSet(ADR(Timeout),500,TRUE);
				TFCommandCase(ADR(CmdExe),100,CommandCase_JMP);

			1: TFCommandCase(ADR(CmdExe),100,CommandCase_JMP);
			(* Case 100 *)
			100:TFStateUpdate(ADR(State),StatePOWER_END);
				TFCommandExeClear(ADR(CmdExe));

			ELSE
				TFError(ErrNOCMDCASE,ErrNULL,ADR(CmdExe),ADR(State),ADR(Error),ADR(ErrorLog));
		END_CASE
	
	(* ******************************************************************************************************** *)
	(* Home *)
	(* ******************************************************************************************************** *)
	CmdHOME:
		CASE CmdExe.CmdCase OF

			(* Case 0 *)
			0: 	TFStateUpdate(ADR(State),StateHOME_RUN);
				TFTimerSet(ADR(Timeout),3000+200,TRUE);
				TFTimerSet(ADR(Timer),3000,TRUE);
				IF NOT IN_SimulazioneSenzaHW THEN
					TFCommandCase(ADR(CmdExe),1,CommandCase_INC);
				ELSE
					TFCommandCase(ADR(CmdExe),100,CommandCase_JMP);
				END_IF

			(* Case 1 - *)
			1: 
				TFCommandCase(ADR(CmdExe),10,CommandCase_JMP);

			(* Case 10 - Set automatico Soglie *)
			10:
				AspirazioneDX1^.Command^.Aspirazione_ON_ScritturaSoglia 	:= TRUE;
				AspirazioneSX1^.Command^.Aspirazione_ON_ScritturaSoglia 	:= TRUE;
				AspirazioneDX2^.Command^.Aspirazione_ON_ScritturaSoglia 	:= TRUE;
				AspirazioneSX2^.Command^.Aspirazione_ON_ScritturaSoglia 	:= TRUE;
				IF AspirazioneDX1^.Status.CommandDone AND AspirazioneSX1^.Status.CommandDone AND
					AspirazioneDX2^.Status.CommandDone AND AspirazioneSX2^.Status.CommandDone THEN
						TFClearAllCmdModulePinzaMagazzino(AspirazioneDX1,AspirazioneSX1,AspirazioneDX2,AspirazioneSX2,CilindroSbloccoRotazione,CilindroSbloccoBascolante);
						TFCommandCase(ADR(CmdExe),100,CommandCase_JMP);
				ELSIF TFTimerDone(ADR(Timer)) THEN
					TFClearAllCmdModulePinzaMagazzino(AspirazioneDX1,AspirazioneSX1,AspirazioneDX2,AspirazioneSX2,CilindroSbloccoRotazione,CilindroSbloccoBascolante);
					TFError(ErrTOHOME,ErrNULL,ADR(CmdExe),ADR(State),ADR(Error),ADR(ErrorLog));
				END_IF
			
	
			(* Case 100 *)
			100:TFStateUpdate(ADR(State),StateHOME_END);
				TFCommandExeClear(ADR(CmdExe));

			ELSE
				TFError(ErrNOCMDCASE,ErrNULL,ADR(CmdExe),ADR(State),ADR(Error),ADR(ErrorLog));
		END_CASE;
		
		IF AspirazioneDX1^.Status.ErrorID <> ErrNULL AND NOT IN_SimulazioneSenzaHW THEN
			TFClearAllCmdModulePinzaMagazzino(AspirazioneDX1,AspirazioneSX1,AspirazioneDX2,AspirazioneSX2,CilindroSbloccoRotazione,CilindroSbloccoBascolante);
			TFError(ErrCYLINDER,AspirazioneDX1^.Status.ErrorID,ADR(CmdExe),ADR(State),ADR(Error),ADR(ErrorLog));
		ELSIF AspirazioneSX1^.Status.ErrorID <> ErrNULL AND NOT IN_SimulazioneSenzaHW THEN
			TFClearAllCmdModulePinzaMagazzino(AspirazioneDX1,AspirazioneSX1,AspirazioneDX2,AspirazioneSX2,CilindroSbloccoRotazione,CilindroSbloccoBascolante);
			TFError(ErrCYLINDER,AspirazioneSX1^.Status.ErrorID,ADR(CmdExe),ADR(State),ADR(Error),ADR(ErrorLog));
		ELSIF AspirazioneDX2^.Status.ErrorID <> ErrNULL AND NOT IN_SimulazioneSenzaHW THEN
			TFClearAllCmdModulePinzaMagazzino(AspirazioneDX1,AspirazioneSX1,AspirazioneDX2,AspirazioneSX2,CilindroSbloccoRotazione,CilindroSbloccoBascolante);
			TFError(ErrCYLINDER,AspirazioneDX2^.Status.ErrorID,ADR(CmdExe),ADR(State),ADR(Error),ADR(ErrorLog));
		ELSIF AspirazioneSX2^.Status.ErrorID <> ErrNULL AND NOT IN_SimulazioneSenzaHW THEN
			TFClearAllCmdModulePinzaMagazzino(AspirazioneDX1,AspirazioneSX1,AspirazioneDX2,AspirazioneSX2,CilindroSbloccoRotazione,CilindroSbloccoBascolante);
			TFError(ErrCYLINDER,AspirazioneSX2^.Status.ErrorID,ADR(CmdExe),ADR(State),ADR(Error),ADR(ErrorLog));
		ELSIF CilindroSbloccoRotazione^.Status.ErrorID <> ErrNULL THEN
			TFClearAllCmdModulePinzaMagazzino(AspirazioneDX1,AspirazioneSX1,AspirazioneDX2,AspirazioneSX2,CilindroSbloccoRotazione,CilindroSbloccoBascolante);
			TFError(ErrCYLINDER,CilindroSbloccoRotazione^.Status.ErrorID,ADR(CmdExe),ADR(State),ADR(Error),ADR(ErrorLog));
		ELSIF TFTimerDone(ADR(Timeout)) THEN
			TFClearAllCmdModulePinzaMagazzino(AspirazioneDX1,AspirazioneSX1,AspirazioneDX2,AspirazioneSX2,CilindroSbloccoRotazione,CilindroSbloccoBascolante);
			TFError(ErrCMDTIMEOUT,ErrNULL,ADR(CmdExe),ADR(State),ADR(Error),ADR(ErrorLog));
		END_IF

	(* ******************************************************************************************************** *)
	(* Manual *)
	(* ******************************************************************************************************** *)
	CmdMAN:
		CASE CmdExe.CmdCase OF
			(* Case 0 *)
			0: 	TFStateUpdate(ADR(State),StateMAN_RUN);
				TFTimerSet(ADR(Timeout),3000,TRUE);
				TFTimerSet(ADR(Timer),10,TRUE);
				IF TFCommandParRead(CmdExe.Cmd.Parameter,ADR(ParametersArray),2) THEN
					MAN_Actuator	:= STRING_TO_UINT(ParametersArray.Parameters[0]);
					MAN_Cmd		:= STRING_TO_UINT(ParametersArray.Parameters[1]);
				ELSE
					TFError(ErrCMDPARNUM,ErrNULL,ADR(CmdExe),ADR(State),ADR(Error),ADR(ErrorLog));
					RETURN;
				END_IF;

				CASE MAN_Actuator OF
					(* Case 0..99 for Actuators *)
					(* Case 100..199  for Axis *)

					(* Case Nop *)
					0:	;

					(* Case 1: *)
					1:	CASE MAN_Cmd OF
							0:	;
							
							
							(* Case 20: Sgancio Sblocco Rotazione *)
							20:	
								CilindroSbloccoRotazione^.Command.Activation 	:= TRUE;
								CilindroSbloccoRotazione^.Command.Deactivation 	:= FALSE;
								TFTimerSet(ADR(Timeout),3000,TRUE);
								TFCommandCase(ADR(CmdExe),20,CommandCase_JMP);
								
							(* Case 21: Aggancio Sblocco Rotazione *)
							21:	
								CilindroSbloccoRotazione^.Command.Activation 	:= FALSE;
								CilindroSbloccoRotazione^.Command.Deactivation 	:= TRUE;
								TFTimerSet(ADR(Timeout),3000,TRUE);
								TFCommandCase(ADR(CmdExe),20,CommandCase_JMP);
	
							(* Case 50: Ativazione Aspirazione SX *)
							50:	
								
								IF NOT IN_SimulazioneSenzaHW THEN 
									AspirazioneSX1^.Command^.Aspirazione_ON		:= TRUE;
									AspirazioneSX1^.Command^.Aspirazione_OFF 	:= FALSE;
									AspirazioneDX1^.Command^.Aspirazione_ON 	:= TRUE;
									AspirazioneDX1^.Command^.Aspirazione_OFF 	:= FALSE;
									AspirazioneSX2^.Command^.Aspirazione_ON 	:= TRUE;
									AspirazioneSX2^.Command^.Aspirazione_OFF 	:= FALSE;
									AspirazioneDX2^.Command^.Aspirazione_ON 	:= TRUE;
									AspirazioneDX2^.Command^.Aspirazione_OFF 	:= FALSE;
	
									TFTimerSet(ADR(Timeout),3000,TRUE);
									TFCommandCase(ADR(CmdExe),50,CommandCase_JMP);
								ELSE
									TFCommandCase(ADR(CmdExe),1,CommandCase_JMP);
								END_IF
										
							(* Case 51: Disattivazione Aspirazione SX *)
							51:	
								StatoPinza.ElementoPrelevato := FALSE;
								IF NOT IN_SimulazioneSenzaHW THEN 
									AspirazioneSX1^.Command^.Aspirazione_ON 	:= FALSE;
									AspirazioneSX1^.Command^.Aspirazione_OFF 	:= TRUE;
									AspirazioneDX1^.Command^.Aspirazione_ON 	:= FALSE;
									AspirazioneDX1^.Command^.Aspirazione_OFF 	:= TRUE;
									AspirazioneSX2^.Command^.Aspirazione_ON 	:= FALSE;
									AspirazioneSX2^.Command^.Aspirazione_OFF 	:= TRUE;
									AspirazioneDX2^.Command^.Aspirazione_ON 	:= FALSE;
									AspirazioneDX2^.Command^.Aspirazione_OFF 	:= TRUE;
									TFTimerSet(ADR(Timeout),3000,TRUE);
									TFCommandCase(ADR(CmdExe),50,CommandCase_JMP);
								ELSE
									TFCommandCase(ADR(CmdExe),1,CommandCase_JMP);
								END_IF

							(* Case 60: Ativazione Aspirazione DX *)
							60:	
								IF NOT IN_SimulazioneSenzaHW THEN 
									AspirazioneSX1^.Command^.Aspirazione_ON 	:= TRUE;
									AspirazioneSX1^.Command^.Aspirazione_OFF 	:= FALSE;
									AspirazioneDX1^.Command^.Aspirazione_ON 	:= TRUE;
									AspirazioneDX1^.Command^.Aspirazione_OFF 	:= FALSE;
									AspirazioneSX2^.Command^.Aspirazione_ON 	:= TRUE;
									AspirazioneSX2^.Command^.Aspirazione_OFF 	:= FALSE;
									AspirazioneDX2^.Command^.Aspirazione_ON 	:= TRUE;
									AspirazioneDX2^.Command^.Aspirazione_OFF 	:= FALSE;
									TFTimerSet(ADR(Timeout),3000,TRUE);
									TFCommandCase(ADR(CmdExe),60,CommandCase_JMP);
								ELSE
									TFCommandCase(ADR(CmdExe),1,CommandCase_JMP);
								END_IF

							(* Case 61: Disattivazione Aspirazione SX *)
							61:	
								StatoPinza.ElementoPrelevato := FALSE;
								IF NOT IN_SimulazioneSenzaHW THEN 
									AspirazioneDX1^.Command^.Aspirazione_ON  := FALSE;
									AspirazioneDX1^.Command^.Aspirazione_OFF := TRUE;
									AspirazioneSX1^.Command^.Aspirazione_ON  := FALSE;
									AspirazioneSX1^.Command^.Aspirazione_OFF := TRUE;
									AspirazioneDX2^.Command^.Aspirazione_ON  := FALSE;
									AspirazioneDX2^.Command^.Aspirazione_OFF := TRUE;
									AspirazioneSX2^.Command^.Aspirazione_ON  := FALSE;
									AspirazioneSX2^.Command^.Aspirazione_OFF := TRUE;
									StatoPinza.ElementoPrelevato := FALSE;
									TFTimerSet(ADR(Timeout),3000,TRUE);
									TFCommandCase(ADR(CmdExe),60,CommandCase_JMP);
								ELSE
									TFCommandCase(ADR(CmdExe),1,CommandCase_JMP);
								END_IF
							ELSE
								TFError(ErrNOCMDCASE,ErrNULL,ADR(CmdExe),ADR(State),ADR(Error),ADR(ErrorLog));
						END_CASE;

					100:CASE MAN_Cmd OF
							0:	;
							ELSE
								TFError(ErrNOCMDCASE,ErrNULL,ADR(CmdExe),ADR(State),ADR(Error),ADR(ErrorLog));
						END_CASE;

					ELSE
						TFError(ErrNOCMDCASE,ErrNULL,ADR(CmdExe),ADR(State),ADR(Error),ADR(ErrorLog));
				END_CASE;

				//IF CmdExe.CmdCase = 0 THEN
					//TFCommandCase(ADR(CmdExe),1,CommandCase_INC);
				//END_IF

			(* Case 1 - *)
			1: 	IF (MAN_Cmd = 0) OR TFTimerDone(ADR(Timer)) THEN
					(* Clear All Output Here *)
					;
					TFStateUpdate(ADR(State),StateMAN_END);
					TFCommandExeClear(ADR(CmdExe));
				END_IF;

			(* Case 20 - CilindroSbloccoRotazione *)
			20: 
				IF CilindroSbloccoRotazione^.Status.Inactive AND CilindroSbloccoRotazione^.Command.Deactivation OR
					CilindroSbloccoRotazione^.Status.Active AND CilindroSbloccoRotazione^.Command.Activation THEN
						CilindroSbloccoRotazione^.Command.Activation 	:= FALSE;
						CilindroSbloccoRotazione^.Command.Deactivation 	:= FALSE;
						TFCommandCase(ADR(CmdExe),100,CommandCase_JMP);
				ELSIF CilindroSbloccoRotazione^.Status.ErrorID <> ErrNULL THEN
					TFClearAllCmdModulePinzaMagazzino(AspirazioneDX1,AspirazioneSX1,AspirazioneDX2,AspirazioneSX2,CilindroSbloccoRotazione,CilindroSbloccoBascolante);
					TFError(ErrCYLINDER,CilindroSbloccoRotazione^.Status.ErrorID,ADR(CmdExe),ADR(State),ADR(Error),ADR(ErrorLog));
				END_IF

			(* Case 50 - AspirazioneSX *)
			50: 
				IF AspirazioneSX1^.Status.CommandDone AND AspirazioneDX1^.Status.CommandDone AND
					AspirazioneSX2^.Status.CommandDone AND AspirazioneDX2^.Status.CommandDone THEN
						TFClearAllCmdModulePinzaMagazzino(AspirazioneDX1,AspirazioneSX1,AspirazioneDX2,AspirazioneSX2,CilindroSbloccoRotazione,CilindroSbloccoBascolante);
						TFCommandCase(ADR(CmdExe),100,CommandCase_JMP);
				ELSIF AspirazioneSX1^.Status.ErrorID <> ErrNULL THEN
					TFClearAllCmdModulePinzaMagazzino(AspirazioneDX1,AspirazioneSX1,AspirazioneDX2,AspirazioneSX2,CilindroSbloccoRotazione,CilindroSbloccoBascolante);
					TFError(ErrCYLINDER,AspirazioneSX1^.Status.ErrorID,ADR(CmdExe),ADR(State),ADR(Error),ADR(ErrorLog));
				ELSIF AspirazioneDX1^.Status.ErrorID <> ErrNULL THEN
					TFClearAllCmdModulePinzaMagazzino(AspirazioneDX1,AspirazioneSX1,AspirazioneDX2,AspirazioneSX2,CilindroSbloccoRotazione,CilindroSbloccoBascolante);
					TFError(ErrCYLINDER,AspirazioneDX1^.Status.ErrorID,ADR(CmdExe),ADR(State),ADR(Error),ADR(ErrorLog));
				ELSIF AspirazioneSX2^.Status.ErrorID <> ErrNULL THEN
					TFClearAllCmdModulePinzaMagazzino(AspirazioneDX1,AspirazioneSX1,AspirazioneDX2,AspirazioneSX2,CilindroSbloccoRotazione,CilindroSbloccoBascolante);
					TFError(ErrCYLINDER,AspirazioneSX2^.Status.ErrorID,ADR(CmdExe),ADR(State),ADR(Error),ADR(ErrorLog));
				ELSIF AspirazioneDX2^.Status.ErrorID <> ErrNULL THEN
					TFClearAllCmdModulePinzaMagazzino(AspirazioneDX1,AspirazioneSX1,AspirazioneDX2,AspirazioneSX2,CilindroSbloccoRotazione,CilindroSbloccoBascolante);
					TFError(ErrCYLINDER,AspirazioneDX2^.Status.ErrorID,ADR(CmdExe),ADR(State),ADR(Error),ADR(ErrorLog));
				END_IF

			(* Case 60 - AspirazioneDX *)
			60: 
				IF AspirazioneSX1^.Status.CommandDone AND AspirazioneDX1^.Status.CommandDone AND
					AspirazioneSX2^.Status.CommandDone AND AspirazioneDX2^.Status.CommandDone THEN
						TFClearAllCmdModulePinzaMagazzino(AspirazioneDX1,AspirazioneSX1,AspirazioneDX2,AspirazioneSX2,CilindroSbloccoRotazione,CilindroSbloccoBascolante);
						TFCommandCase(ADR(CmdExe),100,CommandCase_JMP);
				ELSIF AspirazioneSX1^.Status.ErrorID <> ErrNULL THEN
					TFClearAllCmdModulePinzaMagazzino(AspirazioneDX1,AspirazioneSX1,AspirazioneDX2,AspirazioneSX2,CilindroSbloccoRotazione,CilindroSbloccoBascolante);
					TFError(ErrCYLINDER,AspirazioneSX1^.Status.ErrorID,ADR(CmdExe),ADR(State),ADR(Error),ADR(ErrorLog));
				ELSIF AspirazioneDX1^.Status.ErrorID <> ErrNULL THEN
					TFClearAllCmdModulePinzaMagazzino(AspirazioneDX1,AspirazioneSX1,AspirazioneDX2,AspirazioneSX2,CilindroSbloccoRotazione,CilindroSbloccoBascolante);
					TFError(ErrCYLINDER,AspirazioneDX1^.Status.ErrorID,ADR(CmdExe),ADR(State),ADR(Error),ADR(ErrorLog));
				ELSIF AspirazioneSX2^.Status.ErrorID <> ErrNULL THEN
					TFClearAllCmdModulePinzaMagazzino(AspirazioneDX1,AspirazioneSX1,AspirazioneDX2,AspirazioneSX2,CilindroSbloccoRotazione,CilindroSbloccoBascolante);
					TFError(ErrCYLINDER,AspirazioneSX2^.Status.ErrorID,ADR(CmdExe),ADR(State),ADR(Error),ADR(ErrorLog));
				ELSIF AspirazioneDX2^.Status.ErrorID <> ErrNULL THEN
					TFClearAllCmdModulePinzaMagazzino(AspirazioneDX1,AspirazioneSX1,AspirazioneDX2,AspirazioneSX2,CilindroSbloccoRotazione,CilindroSbloccoBascolante);
					TFError(ErrCYLINDER,AspirazioneDX2^.Status.ErrorID,ADR(CmdExe),ADR(State),ADR(Error),ADR(ErrorLog));
				END_IF

			(* Case 100 - End *)
			100:(* Clear All Output Here *)
				TFStateUpdate(ADR(State),StateMAN_END);
				TFCommandExeClear(ADR(CmdExe));

			ELSE
				TFError(ErrNOCMDCASE,ErrNULL,ADR(CmdExe),ADR(State),ADR(Error),ADR(ErrorLog));
		END_CASE;

		IF TFTimerDone(ADR(Timeout)) THEN
			TFClearAllCmdModulePinzaMagazzino(AspirazioneDX1,AspirazioneSX1,AspirazioneDX2,AspirazioneSX2,CilindroSbloccoRotazione,CilindroSbloccoBascolante);
			TFError(ErrCMDTIMEOUT,ErrNULL,ADR(CmdExe),ADR(State),ADR(Error),ADR(ErrorLog));
		END_IF
	

	(* ******************************************************************************************************** *)
	(* PRELOAD - Attivazione vuoto *)
	(* ******************************************************************************************************** *)
	CmdPRELOAD:
		CASE CmdExe.CmdCase OF
			
			(* Case 0 - Init Command*)
			0: 	TFStateUpdate(ADR(State),StatePRELOAD_RUN);
				TFTimerSet(ADR(Timeout),30000+200,TRUE);
				TFTimerSet(ADR(Timer),30000,TRUE);
				PrelievoSuMagazino := FALSE;
				StatoPinza.ElementoPrelevato := FALSE;
				IF TFCommandParRead(CmdExe.Cmd.Parameter,ADR(ParametersArray),1) THEN
					PrelievoSuMagazino	:= STRING_TO_BOOL(ParametersArray.Parameters[0]);
					IF NOT IN_SimulazioneSenzaHW THEN
						TFCommandCase(ADR(CmdExe),40,CommandCase_JMP);
					ELSE
						TFCommandCase(ADR(CmdExe),100,CommandCase_JMP);
					END_IF
				ELSE
					TFError(ErrCMDPARNUM,ErrNULL,ADR(CmdExe),ADR(State),ADR(Error),ADR(ErrorLog));
					RETURN;
				END_IF;
				
			(* Case 10 - CilindroSbloccoRotazione *)
			10: 
				IF PrelievoSuMagazino AND FALSE THEN
					CilindroSbloccoRotazione^.Command.Activation 	:= AbilitazioneSbloccoRotazione;
					CilindroSbloccoRotazione^.Command.Deactivation 	:= FALSE;
	
					IF (CilindroSbloccoRotazione^.Status.Active OR NOT AbilitazioneSbloccoRotazione)THEN
						CilindroSbloccoRotazione^.Command.Activation 	:= FALSE;
						CilindroSbloccoRotazione^.Command.Deactivation 	:= FALSE;
						TFCommandCase(ADR(CmdExe),40,CommandCase_JMP);
					ELSIF CilindroSbloccoRotazione^.Status.ErrorID <> ErrNULL AND AbilitazioneSbloccoRotazione THEN
						TFClearAllCmdModulePinzaMagazzino(AspirazioneDX1,AspirazioneSX1,AspirazioneDX2,AspirazioneSX2,CilindroSbloccoRotazione,CilindroSbloccoBascolante);
						TFError(ErrCYLINDER,CilindroSbloccoRotazione^.Status.ErrorID,ADR(CmdExe),ADR(State),ADR(Error),ADR(ErrorLog));
					END_IF
				ELSE
					TFCommandCase(ADR(CmdExe),40,CommandCase_JMP);
				END_IF


			(* Case 40 - AspirazioneDX + AspirazioneSX *)
			40: 
				AspirazioneDX1^.Command^.Aspirazione_ON 	:= TRUE;
				AspirazioneDX1^.Command^.Aspirazione_OFF 	:= FALSE;
				AspirazioneSX1^.Command^.Aspirazione_ON 	:= TRUE;
				AspirazioneSX1^.Command^.Aspirazione_OFF 	:= FALSE;
				AspirazioneDX2^.Command^.Aspirazione_ON 	:= TRUE;
				AspirazioneDX2^.Command^.Aspirazione_OFF 	:= FALSE;
				AspirazioneSX2^.Command^.Aspirazione_ON 	:= TRUE;
				AspirazioneSX2^.Command^.Aspirazione_OFF 	:= FALSE;
	
				IF (AspirazioneDX1^.Status.CommandDone AND AspirazioneSX1^.Status.CommandDone AND
					AspirazioneDX2^.Status.CommandDone AND AspirazioneSX2^.Status.CommandDone) OR IN.ByPassSensoreVuoto THEN
						TFClearAllCmdModulePinzaMagazzino(AspirazioneDX1,AspirazioneSX1,AspirazioneDX2,AspirazioneSX2,CilindroSbloccoRotazione,CilindroSbloccoBascolante);
						TFCommandCase(ADR(CmdExe),100,CommandCase_JMP);
				ELSIF AspirazioneSX1^.Status.ErrorID <> ErrNULL AND NOT IN_SimulazioneSenzaHW THEN
					TFClearAllCmdModulePinzaMagazzino(AspirazioneDX1,AspirazioneSX1,AspirazioneDX2,AspirazioneSX2,CilindroSbloccoRotazione,CilindroSbloccoBascolante);
					TFError(ErrCYLINDER,AspirazioneSX1^.Status.ErrorID,ADR(CmdExe),ADR(State),ADR(Error),ADR(ErrorLog));
				ELSIF AspirazioneDX1^.Status.ErrorID <> ErrNULL AND NOT IN_SimulazioneSenzaHW THEN
					TFClearAllCmdModulePinzaMagazzino(AspirazioneDX1,AspirazioneSX1,AspirazioneDX2,AspirazioneSX2,CilindroSbloccoRotazione,CilindroSbloccoBascolante);
					TFError(ErrCYLINDER,AspirazioneDX1^.Status.ErrorID,ADR(CmdExe),ADR(State),ADR(Error),ADR(ErrorLog));
				ELSIF AspirazioneSX2^.Status.ErrorID <> ErrNULL THEN
					TFClearAllCmdModulePinzaMagazzino(AspirazioneDX1,AspirazioneSX1,AspirazioneDX2,AspirazioneSX2,CilindroSbloccoRotazione,CilindroSbloccoBascolante);
					TFError(ErrCYLINDER,AspirazioneSX2^.Status.ErrorID,ADR(CmdExe),ADR(State),ADR(Error),ADR(ErrorLog));
				ELSIF AspirazioneDX2^.Status.ErrorID <> ErrNULL THEN
					TFClearAllCmdModulePinzaMagazzino(AspirazioneDX1,AspirazioneSX1,AspirazioneDX2,AspirazioneSX2,CilindroSbloccoRotazione,CilindroSbloccoBascolante);
					TFError(ErrCYLINDER,AspirazioneDX2^.Status.ErrorID,ADR(CmdExe),ADR(State),ADR(Error),ADR(ErrorLog));
				END_IF
				
			(* Case 100 *)
			100:TFStateUpdate(ADR(State),StatePRELOAD_END);
				TFCommandExeClear(ADR(CmdExe));

			ELSE
				TFError(ErrNOCMDCASE,ErrNULL,ADR(CmdExe),ADR(State),ADR(Error),ADR(ErrorLog));
		END_CASE

		IF TFTimerDone(ADR(Timeout)) THEN
			TFClearAllCmdModulePinzaMagazzino(AspirazioneDX1,AspirazioneSX1,AspirazioneDX2,AspirazioneSX2,CilindroSbloccoRotazione,CilindroSbloccoBascolante);
			TFError(ErrCMDTIMEOUT,ErrNULL,ADR(CmdExe),ADR(State),ADR(Error),ADR(ErrorLog));
		END_IF
	
	(* ******************************************************************************************************** *)
	(* LOAD - Presa del pezzo *)
	(* ******************************************************************************************************** *)
	CmdCHECKPRESENCE:
		CASE CmdExe.CmdCase OF
			
			(* Case 0 - Init Command*)
			0: 	TFStateUpdate(ADR(State),StateCHECKPRESENCE_RUN);
				TFTimerSet(ADR(Timeout),60000.0+100+HMI_TempoControlloPresaPiastrella,TRUE);
				TFTimerSet(ADR(Timer),2000.0+HMI_TempoControlloPresaPiastrella,TRUE);
				TFTimerSet(ADR(TimerPresaPiastrella),HMI_TempoControlloPresaPiastrella,TRUE);
				StatoPinza.ElementoPrelevato := FALSE;

				TFCommandCase(ADR(CmdExe),1,CommandCase_INC);
				
			(* Case 1 - *)					
			1:
				IF IN.ByPassSensoreVuoto OR TFTimerDone(ADR(TimerPresaPiastrella)) THEN 
					//Tutte piastrelle o tutte falde
					IF (AspirazioneDX1^.Status.DepressioneSoglia1_OK AND AspirazioneSX1^.Status.DepressioneSoglia1_OK AND
						 AspirazioneDX2^.Status.DepressioneSoglia1_OK AND AspirazioneSX2^.Status.DepressioneSoglia1_OK) OR IN.ByPassSensoreVuoto THEN
						StatoPinza.ElementoPrelevato := TRUE;
						TFCommandCase(ADR(CmdExe),11,CommandCase_JMP);
					ELSIF TFTimerDone(ADR(TimerPresaPiastrella)) THEN
						TFCommandCase(ADR(CmdExe),11,CommandCase_JMP);
						StatoPinza.ElementoPrelevato := IN.ByPassSensoreVuoto;	
					END_IF			
				END_IF
				IF TFTimerDone(ADR(Timer)) THEN
					TFClearAllCmdModulePinzaMagazzino(AspirazioneDX1,AspirazioneSX1,AspirazioneDX2,AspirazioneSX2,CilindroSbloccoRotazione,CilindroSbloccoBascolante);
					TFError(ErrMalfunzionamentoSensoriPresenzaPinza,ErrNULL,ADR(CmdExe),ADR(State),ADR(Error),ADR(ErrorLog));
				ELSIF TFTimerDone(ADR(Timeout)) THEN
					TFClearAllCmdModulePinzaMagazzino(AspirazioneDX1,AspirazioneSX1,AspirazioneDX2,AspirazioneSX2,CilindroSbloccoRotazione,CilindroSbloccoBascolante);
					TFError(ErrCMDTIMEOUT,ErrNULL,ADR(CmdExe),ADR(State),ADR(Error),ADR(ErrorLog));
				END_IF
						
			(* Case 11 - *)		
			11:
				TFStateUpdate(ADR(State),StateCHECKPRESENCE_RUN+10);
				TFCommandCase(ADR(CmdExe),100,CommandCase_JMP);
								
					
			(* Case 100 *)
			100:TFStateUpdate(ADR(State),StateCHECKPRESENCE_END);
				TFCommandExeClear(ADR(CmdExe));

			ELSE
				TFError(ErrNOCMDCASE,ErrNULL,ADR(CmdExe),ADR(State),ADR(Error),ADR(ErrorLog));
		END_CASE

	(* ******************************************************************************************************** *)
	(* CmdSbloccaBascolante - SGANCIO BASCULANTE *)
	(* ******************************************************************************************************** *)
	CmdSbloccaBascolante:
		CASE CmdExe.CmdCase OF
			
			(* Case 0 - Init Command*)
			0: 	TFStateUpdate(ADR(State),StateSbloccaBascolante_RUN);
				TFTimerSet(ADR(Timeout),30000+200,TRUE);
				TFTimerSet(ADR(Timer),30000,TRUE);
				IF NOT IN_SimulazioneSenzaHW THEN
					TFCommandCase(ADR(CmdExe),10,CommandCase_JMP);
				ELSE
					TFCommandCase(ADR(CmdExe),100,CommandCase_JMP);
				END_IF
				
			(* Case 10 - CilindroSblocco bacolante *)
			10: 
				CilindroSbloccoBascolante^.Command.Activation 	:= AbilitazioneSbloccoBascolante;
				CilindroSbloccoBascolante^.Command.Deactivation := FALSE;

				IF (CilindroSbloccoBascolante^.Status.Active OR NOT AbilitazioneSbloccoBascolante)THEN
					CilindroSbloccoBascolante^.Command.Activation 	:= FALSE;
					CilindroSbloccoBascolante^.Command.Deactivation 	:= FALSE;
					TFCommandCase(ADR(CmdExe),100,CommandCase_JMP);
				ELSIF CilindroSbloccoBascolante^.Status.ErrorID <> ErrNULL AND AbilitazioneSbloccoBascolante THEN
					TFClearAllCmdModulePinzaMagazzino(AspirazioneDX1,AspirazioneSX1,AspirazioneDX2,AspirazioneSX2,CilindroSbloccoRotazione,CilindroSbloccoBascolante);
					TFError(ErrCYLINDER,CilindroSbloccoBascolante^.Status.ErrorID,ADR(CmdExe),ADR(State),ADR(Error),ADR(ErrorLog));
				END_IF

				
			(* Case 100 *)
			100:TFStateUpdate(ADR(State),StateSbloccaBascolante_END);
				TFCommandExeClear(ADR(CmdExe));

			ELSE
				TFError(ErrNOCMDCASE,ErrNULL,ADR(CmdExe),ADR(State),ADR(Error),ADR(ErrorLog));
		END_CASE

		IF TFTimerDone(ADR(Timeout)) THEN
			TFClearAllCmdModulePinzaMagazzino(AspirazioneDX1,AspirazioneSX1,AspirazioneDX2,AspirazioneSX2,CilindroSbloccoRotazione,CilindroSbloccoBascolante);
			TFError(ErrCMDTIMEOUT,ErrNULL,ADR(CmdExe),ADR(State),ADR(Error),ADR(ErrorLog));
		END_IF
		
		(* ******************************************************************************************************** *)
	(* CmdBloccaBascolante - AGGANCIO BASCULANTE *)
	(* ******************************************************************************************************** *)
	CmdBloccaBascolante:
		CASE CmdExe.CmdCase OF
			
			(* Case 0 - Init Command*)
			0: 	TFStateUpdate(ADR(State),StateBloccaBascolante_RUN);
				TFTimerSet(ADR(Timeout),30000+200,TRUE);
				TFTimerSet(ADR(Timer),30000,TRUE);
				IF NOT IN_SimulazioneSenzaHW THEN
					TFCommandCase(ADR(CmdExe),10,CommandCase_JMP);
				ELSE
					TFCommandCase(ADR(CmdExe),100,CommandCase_JMP);
				END_IF
				
			(* Case 10 - CilindroSblocco bacolante *)
			10: 
				CilindroSbloccoBascolante^.Command.Activation 	:= FALSE;
				CilindroSbloccoBascolante^.Command.Deactivation := TRUE;

				IF  CilindroSbloccoBascolante^.Status.Inactive THEN
					CilindroSbloccoBascolante^.Command.Activation 	:= FALSE;
					CilindroSbloccoBascolante^.Command.Deactivation := FALSE;
					TFCommandCase(ADR(CmdExe),100,CommandCase_JMP);
				ELSIF CilindroSbloccoBascolante^.Status.ErrorID <> ErrNULL AND AbilitazioneSbloccoBascolante THEN
					TFClearAllCmdModulePinzaMagazzino(AspirazioneDX1,AspirazioneSX1,AspirazioneDX2,AspirazioneSX2,CilindroSbloccoRotazione,CilindroSbloccoBascolante);
					TFError(ErrCYLINDER,CilindroSbloccoBascolante^.Status.ErrorID,ADR(CmdExe),ADR(State),ADR(Error),ADR(ErrorLog));
				END_IF

				
			(* Case 100 *)
			100:TFStateUpdate(ADR(State),StateBloccaBascolante_END);
				TFCommandExeClear(ADR(CmdExe));

			ELSE
				TFError(ErrNOCMDCASE,ErrNULL,ADR(CmdExe),ADR(State),ADR(Error),ADR(ErrorLog));
		END_CASE

		IF TFTimerDone(ADR(Timeout)) THEN
			TFClearAllCmdModulePinzaMagazzino(AspirazioneDX1,AspirazioneSX1,AspirazioneDX2,AspirazioneSX2,CilindroSbloccoRotazione,CilindroSbloccoBascolante);
			TFError(ErrCMDTIMEOUT,ErrNULL,ADR(CmdExe),ADR(State),ADR(Error),ADR(ErrorLog));
		END_IF
		
	(* ******************************************************************************************************** *)
	(* CmdSbloccaRotazione - SGANCIO rotazione *)
	(* ******************************************************************************************************** *)
	CmdSbloccaRotazione:
		CASE CmdExe.CmdCase OF
			
			(* Case 0 - Init Command*)
			0: 	TFStateUpdate(ADR(State),StateSbloccaRotazione_RUN);
				TFTimerSet(ADR(Timeout),30000+200,TRUE);
				TFTimerSet(ADR(Timer),30000,TRUE);
				IF NOT IN_SimulazioneSenzaHW THEN
					TFCommandCase(ADR(CmdExe),10,CommandCase_JMP);
				ELSE
					TFCommandCase(ADR(CmdExe),100,CommandCase_JMP);
				END_IF
				
			(* Case 10 - CilindroSblocco bacolante *)
			10: 
				CilindroSbloccoRotazione^.Command.Activation 	:= AbilitazioneSbloccoRotazione;
				CilindroSbloccoRotazione^.Command.Deactivation := FALSE;

				IF (CilindroSbloccoRotazione^.Status.Active OR NOT AbilitazioneSbloccoRotazione)THEN
					CilindroSbloccoRotazione^.Command.Activation 	:= FALSE;
					CilindroSbloccoRotazione^.Command.Deactivation 	:= FALSE;
					TFCommandCase(ADR(CmdExe),100,CommandCase_JMP);
				ELSIF CilindroSbloccoBascolante^.Status.ErrorID <> ErrNULL AND AbilitazioneSbloccoRotazione THEN
					TFClearAllCmdModulePinzaMagazzino(AspirazioneDX1,AspirazioneSX1,AspirazioneDX2,AspirazioneSX2,CilindroSbloccoRotazione,CilindroSbloccoBascolante);
					TFError(ErrCYLINDER,CilindroSbloccoRotazione^.Status.ErrorID,ADR(CmdExe),ADR(State),ADR(Error),ADR(ErrorLog));
				END_IF

				
			(* Case 100 *)
			100:TFStateUpdate(ADR(State),StateSbloccaRotazione_END);
				TFCommandExeClear(ADR(CmdExe));

			ELSE
				TFError(ErrNOCMDCASE,ErrNULL,ADR(CmdExe),ADR(State),ADR(Error),ADR(ErrorLog));
		END_CASE

		IF TFTimerDone(ADR(Timeout)) THEN
			TFClearAllCmdModulePinzaMagazzino(AspirazioneDX1,AspirazioneSX1,AspirazioneDX2,AspirazioneSX2,CilindroSbloccoRotazione,CilindroSbloccoBascolante);
			TFError(ErrCMDTIMEOUT,ErrNULL,ADR(CmdExe),ADR(State),ADR(Error),ADR(ErrorLog));
		END_IF
		
	(* ******************************************************************************************************** *)
	(* CmdBloccaROTAZIONE - BLOCCA ROTAZIONE *)
	(* ******************************************************************************************************** *)
	CmdBloccaRotazione:
		CASE CmdExe.CmdCase OF
			
			(* Case 0 - Init Command*)
			0: 	TFStateUpdate(ADR(State),StateBloccaRotazione_RUN);
				TFTimerSet(ADR(Timeout),30000+200,TRUE);
				TFTimerSet(ADR(Timer),30000,TRUE);
				IF NOT IN_SimulazioneSenzaHW THEN
					TFCommandCase(ADR(CmdExe),10,CommandCase_JMP);
				ELSE
					TFCommandCase(ADR(CmdExe),100,CommandCase_JMP);
				END_IF
				
			(* Case 10 - CilindroSblocco bacolante *)
			10: 
				CilindroSbloccoRotazione^.Command.Activation 	:= FALSE;
				CilindroSbloccoRotazione^.Command.Deactivation  := TRUE;

				IF (CilindroSbloccoRotazione^.Status.Inactive) THEN
					CilindroSbloccoRotazione^.Command.Activation 	:= FALSE;
					CilindroSbloccoRotazione^.Command.Deactivation := FALSE;
					TFCommandCase(ADR(CmdExe),100,CommandCase_JMP);
				ELSIF CilindroSbloccoBascolante^.Status.ErrorID <> ErrNULL THEN
					TFClearAllCmdModulePinzaMagazzino(AspirazioneDX1,AspirazioneSX1,AspirazioneDX2,AspirazioneSX2,CilindroSbloccoRotazione,CilindroSbloccoBascolante);
					TFError(ErrCYLINDER,CilindroSbloccoBascolante^.Status.ErrorID,ADR(CmdExe),ADR(State),ADR(Error),ADR(ErrorLog));
				END_IF

				
			(* Case 100 *)
			100:TFStateUpdate(ADR(State),StateBloccaBascolante_END);
				TFCommandExeClear(ADR(CmdExe));

			ELSE
				TFError(ErrNOCMDCASE,ErrNULL,ADR(CmdExe),ADR(State),ADR(Error),ADR(ErrorLog));
		END_CASE

		IF TFTimerDone(ADR(Timeout)) THEN
			TFClearAllCmdModulePinzaMagazzino(AspirazioneDX1,AspirazioneSX1,AspirazioneDX2,AspirazioneSX2,CilindroSbloccoRotazione,CilindroSbloccoBascolante);
			TFError(ErrCMDTIMEOUT,ErrNULL,ADR(CmdExe),ADR(State),ADR(Error),ADR(ErrorLog));
		END_IF
		
	(* ******************************************************************************************************** *)
	(* CmdBloccaPinza- BLOCCA ROTAZIONE + BLOCCA BASCULANTE *)
	(* ******************************************************************************************************** *)
	CmdBloccaPinza:
		CASE CmdExe.CmdCase OF
			
			(* Case 0 - Init Command*)
			0: 	TFStateUpdate(ADR(State),StateBloccaPinza_RUN);
				TFTimerSet(ADR(Timeout),30000+200,TRUE);
				TFTimerSet(ADR(Timer),30000,TRUE);
				IF NOT IN_SimulazioneSenzaHW THEN
					TFCommandCase(ADR(CmdExe),10,CommandCase_JMP);
				ELSE
					TFCommandCase(ADR(CmdExe),100,CommandCase_JMP);
				END_IF
				
			(* Case 10 - CilindroSblocco bascolante + rotazione *)
			10: 
				CilindroSbloccoRotazione^.Command.Activation 	:= FALSE;
				CilindroSbloccoRotazione^.Command.Deactivation  := TRUE;
				
				CilindroSbloccoBascolante^.Command.Activation 	:= FALSE;
				CilindroSbloccoBascolante^.Command.Deactivation  := TRUE;

				IF (CilindroSbloccoRotazione^.Status.Inactive) AND CilindroSbloccoRotazione^.Status.Inactive THEN
					CilindroSbloccoRotazione^.Command.Activation 	:= FALSE;
					CilindroSbloccoRotazione^.Command.Deactivation := FALSE;
					CilindroSbloccoBascolante^.Command.Activation 	:= FALSE;
					CilindroSbloccoBascolante^.Command.Deactivation  := FALSE;

					TFCommandCase(ADR(CmdExe),100,CommandCase_JMP);
				ELSIF CilindroSbloccoBascolante^.Status.ErrorID <> ErrNULL THEN
					TFClearAllCmdModulePinzaMagazzino(AspirazioneDX1,AspirazioneSX1,AspirazioneDX2,AspirazioneSX2,CilindroSbloccoRotazione,CilindroSbloccoBascolante);
					TFError(ErrCYLINDER,CilindroSbloccoBascolante^.Status.ErrorID,ADR(CmdExe),ADR(State),ADR(Error),ADR(ErrorLog));
				ELSIF CilindroSbloccoRotazione^.Status.ErrorID <> ErrNULL THEN
					TFClearAllCmdModulePinzaMagazzino(AspirazioneDX1,AspirazioneSX1,AspirazioneDX2,AspirazioneSX2,CilindroSbloccoRotazione,CilindroSbloccoBascolante);
					TFError(ErrCYLINDER,CilindroSbloccoRotazione^.Status.ErrorID,ADR(CmdExe),ADR(State),ADR(Error),ADR(ErrorLog));
				END_IF

				
			(* Case 100 *)
			100:TFStateUpdate(ADR(State),StateBloccaPinza_END);
				TFCommandExeClear(ADR(CmdExe));

			ELSE
				TFError(ErrNOCMDCASE,ErrNULL,ADR(CmdExe),ADR(State),ADR(Error),ADR(ErrorLog));
		END_CASE

		IF TFTimerDone(ADR(Timeout)) THEN
			TFClearAllCmdModulePinzaMagazzino(AspirazioneDX1,AspirazioneSX1,AspirazioneDX2,AspirazioneSX2,CilindroSbloccoRotazione,CilindroSbloccoBascolante);
			TFError(ErrCMDTIMEOUT,ErrNULL,ADR(CmdExe),ADR(State),ADR(Error),ADR(ErrorLog));
		END_IF

	
	(* ******************************************************************************************************** *)
	(* CmdSbloccaPinza- SBLOCCA ROTAZIONE + SBLOCCA BASCULANTE *)
	(* ******************************************************************************************************** *)
	CmdSbloccaPinza:
			CASE CmdExe.CmdCase OF
				
				(* Case 0 - Init Command*)
				0: 	TFStateUpdate(ADR(State),StateSbloccaPinza_RUN);
					TFTimerSet(ADR(Timeout),30000+200,TRUE);
					TFTimerSet(ADR(Timer),30000,TRUE);
					IF NOT IN_SimulazioneSenzaHW THEN
						TFCommandCase(ADR(CmdExe),10,CommandCase_JMP);
					ELSE
						TFCommandCase(ADR(CmdExe),100,CommandCase_JMP);
					END_IF
					
				(* Case 10 - CilindroSblocco bascolante + rotazione *)
				10: 
					CilindroSbloccoBascolante^.Command.Activation 	:= AbilitazioneSbloccoBascolante;
					CilindroSbloccoBascolante^.Command.Deactivation := FALSE;
					CilindroSbloccoRotazione^.Command.Activation 	:= AbilitazioneSbloccoRotazione;
					CilindroSbloccoRotazione^.Command.Deactivation  := FALSE;
	
					IF (CilindroSbloccoBascolante^.Status.Active OR NOT AbilitazioneSbloccoBascolante) AND 
						(CilindroSbloccoRotazione^.Status.Active OR NOT AbilitazioneSbloccoRotazione) THEN
							CilindroSbloccoBascolante^.Command.Activation 	:= FALSE;
							CilindroSbloccoBascolante^.Command.Deactivation := FALSE;
							CilindroSbloccoRotazione^.Command.Activation 	:= FALSE;
							CilindroSbloccoRotazione^.Command.Deactivation  := FALSE;
							TFCommandCase(ADR(CmdExe),100,CommandCase_JMP);
					ELSIF CilindroSbloccoBascolante^.Status.ErrorID <> ErrNULL AND AbilitazioneSbloccoBascolante THEN
						TFClearAllCmdModulePinzaMagazzino(AspirazioneDX1,AspirazioneSX1,AspirazioneDX2,AspirazioneSX2,CilindroSbloccoRotazione,CilindroSbloccoBascolante);
						TFError(ErrCYLINDER,CilindroSbloccoBascolante^.Status.ErrorID,ADR(CmdExe),ADR(State),ADR(Error),ADR(ErrorLog));
					ELSIF CilindroSbloccoRotazione^.Status.ErrorID <> ErrNULL THEN
						TFClearAllCmdModulePinzaMagazzino(AspirazioneDX1,AspirazioneSX1,AspirazioneDX2,AspirazioneSX2,CilindroSbloccoRotazione,CilindroSbloccoBascolante);
						TFError(ErrCYLINDER,CilindroSbloccoRotazione^.Status.ErrorID,ADR(CmdExe),ADR(State),ADR(Error),ADR(ErrorLog));
					END_IF
					
				(* Case 100 *)
				100:TFStateUpdate(ADR(State),StateSbloccaPinza_END);
					TFCommandExeClear(ADR(CmdExe));
	
				ELSE
					TFError(ErrNOCMDCASE,ErrNULL,ADR(CmdExe),ADR(State),ADR(Error),ADR(ErrorLog));
			END_CASE
	
			IF TFTimerDone(ADR(Timeout)) THEN
				TFClearAllCmdModulePinzaMagazzino(AspirazioneDX1,AspirazioneSX1,AspirazioneDX2,AspirazioneSX2,CilindroSbloccoRotazione,CilindroSbloccoBascolante);
				TFError(ErrCMDTIMEOUT,ErrNULL,ADR(CmdExe),ADR(State),ADR(Error),ADR(ErrorLog));
			END_IF
		
	
	(* ******************************************************************************************************** *)
	(* UNLOAD - Attivazione aspirazione + discesa ventose *)
	(* ******************************************************************************************************** *)
	CmdUNLOAD:
		CASE CmdExe.CmdCase OF
			
			(* Case 0 - Init Command*)
			0: 	TFStateUpdate(ADR(State),StateUNLOAD_RUN);
				TFTimerSet(ADR(Timeout),30000+200,TRUE);
				TFTimerSet(ADR(Timer),30000,TRUE);
				DisattivazioneTotaleAspirazioni := FALSE;
				ByPassAttesaDistacco := FALSE;
				IF NOT IN_SimulazioneSenzaHW THEN
					TFCommandCase(ADR(CmdExe),20,CommandCase_JMP);
				ELSE
					TFCommandCase(ADR(CmdExe),100,CommandCase_JMP);
				END_IF
			
			(* Case 20 - Disattivazione aspirazione piastrella *)		
			20: 
				AspirazioneDX1^.Command^.Aspirazione_ON 	:= FALSE;
				AspirazioneDX1^.Command^.Aspirazione_OFF 	:= TRUE;
				AspirazioneSX1^.Command^.Aspirazione_ON 	:= FALSE;
				AspirazioneSX1^.Command^.Aspirazione_OFF 	:= TRUE;
				AspirazioneDX2^.Command^.Aspirazione_ON 	:= FALSE;
				AspirazioneDX2^.Command^.Aspirazione_OFF 	:= TRUE;
				AspirazioneSX2^.Command^.Aspirazione_ON 	:= FALSE;
				AspirazioneSX2^.Command^.Aspirazione_OFF 	:= TRUE;
				IF NOT AspirazioneDX1^.Status.DepressioneSoglia1_OK AND NOT AspirazioneDX1^.Status.DepressioneSoglia1_OK AND
					NOT AspirazioneDX1^.Status.DepressioneSoglia1_OK AND NOT AspirazioneDX1^.Status.DepressioneSoglia1_OK THEN
						ByPassAttesaDistacco := TRUE;
				END_IF
				
				IF AspirazioneDX1^.Status.CommandDone AND AspirazioneSX1^.Status.CommandDone AND
					AspirazioneDX2^.Status.CommandDone AND AspirazioneSX2^.Status.CommandDone THEN
						TFClearAllCmdModulePinzaMagazzino(AspirazioneDX1,AspirazioneSX1,AspirazioneDX2,AspirazioneSX2,CilindroSbloccoRotazione,CilindroSbloccoBascolante);
						StatoPinza.ElementoPrelevato := FALSE;
						TFTimerSet(ADR(TimerAspirazione),HMI_TempoRilascioInDeposito,TRUE);
						TFCommandCase(ADR(CmdExe),30,CommandCase_JMP);
				ELSIF AspirazioneSX1^.Status.ErrorID <> ErrNULL THEN
					TFClearAllCmdModulePinzaMagazzino(AspirazioneDX1,AspirazioneSX1,AspirazioneDX2,AspirazioneSX2,CilindroSbloccoRotazione,CilindroSbloccoBascolante);
					TFError(ErrCYLINDER,AspirazioneSX1^.Status.ErrorID,ADR(CmdExe),ADR(State),ADR(Error),ADR(ErrorLog));
				ELSIF AspirazioneDX1^.Status.ErrorID <> ErrNULL THEN
					TFClearAllCmdModulePinzaMagazzino(AspirazioneDX1,AspirazioneSX1,AspirazioneDX2,AspirazioneSX2,CilindroSbloccoRotazione,CilindroSbloccoBascolante);
					TFError(ErrCYLINDER,AspirazioneDX1^.Status.ErrorID,ADR(CmdExe),ADR(State),ADR(Error),ADR(ErrorLog));
				END_IF
			
			(* Case 30 - Attesa tempo distacco *)		
			30:
				IF TFTimerDone(ADR(TimerAspirazione)) OR ByPassAttesaDistacco THEN
					IF IN.RichiestaRicalibrazioneOvemEsterna THEN
						IN.RichiestaRicalibrazioneOvemEsterna := FALSE;
						TFCommandCase(ADR(CmdExe),40,CommandCase_JMP);
					ELSE
						TFCommandCase(ADR(CmdExe),100,CommandCase_JMP);
					END_IF		
				END_IF
				
			(* Case 40 - Attesa tempo distacco *)		
			40:	
				AspirazioneDX1^.Command^.Aspirazione_ON_ScritturaSoglia 	:= TRUE;
				AspirazioneSX1^.Command^.Aspirazione_ON_ScritturaSoglia 	:= TRUE;
				AspirazioneDX2^.Command^.Aspirazione_ON_ScritturaSoglia 	:= TRUE;
				AspirazioneSX2^.Command^.Aspirazione_ON_ScritturaSoglia 	:= TRUE;
				IF AspirazioneDX1^.Status.CommandDone AND AspirazioneSX1^.Status.CommandDone AND
					AspirazioneDX2^.Status.CommandDone AND AspirazioneSX2^.Status.CommandDone THEN
						TFClearAllCmdModulePinzaMagazzino(AspirazioneDX1,AspirazioneSX1,AspirazioneDX2,AspirazioneSX2,CilindroSbloccoRotazione,CilindroSbloccoBascolante);
						TFCommandCase(ADR(CmdExe),100,CommandCase_JMP);
				ELSIF TFTimerDone(ADR(Timer)) THEN
					TFClearAllCmdModulePinzaMagazzino(AspirazioneDX1,AspirazioneSX1,AspirazioneDX2,AspirazioneSX2,CilindroSbloccoRotazione,CilindroSbloccoBascolante);
					TFError(ErrTOHOME,ErrNULL,ADR(CmdExe),ADR(State),ADR(Error),ADR(ErrorLog));
				END_IF
				
			(* Case 100 *)
			100:
				StatoPinza.ElementoPrelevato := FALSE;
				TFStateUpdate(ADR(State),StateUNLOAD_END);
				TFCommandExeClear(ADR(CmdExe));

			ELSE
				TFError(ErrNOCMDCASE,ErrNULL,ADR(CmdExe),ADR(State),ADR(Error),ADR(ErrorLog));
		END_CASE

		IF TFTimerDone(ADR(Timeout)) THEN
			TFClearAllCmdModulePinzaMagazzino(AspirazioneDX1,AspirazioneSX1,AspirazioneDX2,AspirazioneSX2,CilindroSbloccoRotazione,CilindroSbloccoBascolante);
			TFError(ErrCMDTIMEOUT,ErrNULL,ADR(CmdExe),ADR(State),ADR(Error),ADR(ErrorLog));
		END_IF

	(* ******************************************************************************************************** *)
	(* POSTUNLOAD - AGGANCIO BASCULANTE *)
	(* ******************************************************************************************************** *)
	CmdPOSTUNLOAD:
		CASE CmdExe.CmdCase OF
			
			(* Case 0 - Init Command*)
			0: 	TFStateUpdate(ADR(State),StatePOSTUNLOAD_RUN);
				TFTimerSet(ADR(Timeout),30000+200,TRUE);
				TFTimerSet(ADR(Timer),30000,TRUE);
				IF NOT IN_SimulazioneSenzaHW THEN
					TFCommandCase(ADR(CmdExe),10,CommandCase_JMP);
				ELSE
					TFCommandCase(ADR(CmdExe),100,CommandCase_JMP);
				END_IF
				
			(* Case 10 - CilindroSbloccoRotazione *)
			10: 
				CilindroSbloccoRotazione^.Command.Activation 	:= FALSE;
				CilindroSbloccoRotazione^.Command.Deactivation 	:= TRUE;

				IF (CilindroSbloccoRotazione^.Status.Inactive)THEN
					CilindroSbloccoRotazione^.Command.Activation 	:= FALSE;
					CilindroSbloccoRotazione^.Command.Deactivation 	:= FALSE;
					TFCommandCase(ADR(CmdExe),100,CommandCase_JMP);
				ELSIF CilindroSbloccoRotazione^.Status.ErrorID <> ErrNULL THEN
					TFClearAllCmdModulePinzaMagazzino(AspirazioneDX1,AspirazioneSX1,AspirazioneDX2,AspirazioneSX2,CilindroSbloccoRotazione,CilindroSbloccoBascolante);
					TFError(ErrCYLINDER,CilindroSbloccoRotazione^.Status.ErrorID,ADR(CmdExe),ADR(State),ADR(Error),ADR(ErrorLog));
				END_IF
			
			(* Case 100 *)
			100:TFStateUpdate(ADR(State),StatePOSTUNLOAD_END);
				TFCommandExeClear(ADR(CmdExe));

			ELSE
				TFError(ErrNOCMDCASE,ErrNULL,ADR(CmdExe),ADR(State),ADR(Error),ADR(ErrorLog));
		END_CASE

		IF TFTimerDone(ADR(Timeout)) THEN
			TFClearAllCmdModulePinzaMagazzino(AspirazioneDX1,AspirazioneSX1,AspirazioneDX2,AspirazioneSX2,CilindroSbloccoRotazione,CilindroSbloccoBascolante);
			TFError(ErrCMDTIMEOUT,ErrNULL,ADR(CmdExe),ADR(State),ADR(Error),ADR(ErrorLog));
		END_IF

	ELSE
		TFError(ErrNOCMD,ErrNULL,ADR(CmdExe),ADR(State),ADR(Error),ADR(ErrorLog));

END_CASE;


(* ******************************************************************************************************** *)
(* State Input/Output *)
(* ******************************************************************************************************** *)
(* Fill Input/Output bit with sensor, electrovalve, etc. status *)

StatoPinza.LatoDxPiastrellaInPresa	:= ((AspirazioneDX1^.Status.DepressioneSoglia1_OK AND AspirazioneDX2^.Status.DepressioneSoglia1_OK)  OR IN.ByPassSensoreVuoto);// AND NOT IN.TastoreCartoneDX;
StatoPinza.LatoSxPiastrellaInPresa	:=((AspirazioneSX1^.Status.DepressioneSoglia1_OK AND AspirazioneSX2^.Status.DepressioneSoglia1_OK)  OR IN.ByPassSensoreVuoto);// AND NOT IN.TastoreCartoneSX;
StatoPinza.RotazioneBloccata		:= CilindroSbloccoRotazione^.Status.Inactive;
StatoPinza.RotazioneSbloccata 		:= CilindroSbloccoRotazione^.Status.Active;
StatoPinza.PianoInPresa				:= StatoPinza.LatoDxPiastrellaInPresa AND StatoPinza.LatoSxPiastrellaInPresa OR (IN.ByPassSensoreVuoto AND StatoPinza.ElementoPrelevato);

(* ******************************************************************************************************** *)
(* Input *)
(* ******************************************************************************************************** *)

(* ******************************************************************************************************** *)
(* Alarm *)
(* ******************************************************************************************************** *)

(* ******************************************************************************************************** *)
(* Error Check - Clear All Output!!! *)
(* ******************************************************************************************************** *)
IF Error.Code > ErrNULL THEN
	IF CmdExe.Code <> CmdNOP THEN
		IF CmdExe.Code <> CmdSTOP AND
			CmdExe.Code <> CmdPOWER AND
			CmdExe.Code <> CmdRESET AND
			CmdExe.Code <> CmdMAN AND
			CmdExe.Code <> CmdLOAD AND
			CmdExe.Code <> CmdUNLOAD THEN
			TFCommandClear(ADR(CmdNext));
			TFCommandExeClear(ADR(CmdExe));

			(* Clear All Output Here *)

		END_IF;
	END_IF;
END_IF;


(* ******************************************************************************************************** *)
(* Common Outputs *)
(* ******************************************************************************************************** *)

END_FUNCTION_BLOCK

// ---- POUs/TFModules/Moduli TF/TFModulePalletizer_Pinza_2Ovem.TcPOU

FUNCTION_BLOCK TFModulePalletizer_Pinza_2Ovem
VAR_INPUT
	Cmd : CommandBuffer;
	Cfg : Config;
	IN : TFMchinePalletizer_PinzaVentose_IN;
		
	IN_Ax : Module_Palletizer_Ax_IN;
	
	AspirazioneDX : POINTER TO TF_VacumOVEM;
	AspirazioneSX : POINTER TO TF_VacumOVEM;

	CilindroApertura 			: POINTER TO DC_Cylinder;
	CilindroSbloccoRotazione 	: POINTER TO SC_Cylinder;
	AspirazioneFaldaDX 			: POINTER TO SC_Cylinder;
	AspirazioneFaldaSX 			: POINTER TO SC_Cylinder;
	
	ModuleJ : POINTER TO TFModulePalletizer_Ax;

	ManCmd 				: POINTER TO TFMachinePalletizer_PinzaVentoseManCmd;
	ElementoInPrelievo 	: TFMachinePalletizer_PlaceElement;
	DataElement			: TFMachinePalletizer_DataElement; (* Struttura dati che la macchina acquisisce/trasferisce in fase di pallettizzazione/depallettizazione *)
	PrelievoSuCavallina : BOOL;//indica che il prelievo è su cavallina
	AbilitazioneCilindriTastatori : bool;

	Mission : POINTER TO TFMachinePalletizer_Mission;
	AbilitazioneSbloccoRotazione 	: BOOL;//Abilitazione sblocco pinza
	AbilitaAperturaAutomaticaPinza : BOOL;//Abilitazione apertura automatica pinza
	PrelivoDaPalletSingoloConFalde : BOOL;
	AbilitaPrioritaPrelPiasterllaPianiSfalsati : bool;
END_VAR
VAR_OUTPUT
	CmdExe : CommandExe;
	CmdExd : CommandExe;
	CmdNext : Command;
	CmdLog : CommandLog;
	ProgramLog : ProgrammaLog; 
	State : State;
	StateLog : StateLog;
	Error : Error;
	ErrorLog : ErrorLog;
	Warning : Warning;
	WarningLog : WarningLog;
	OUT : TFMachinePalletizer_PinzaVentose_OUT;
	StatoPinza : TFMachinePalletizer_PinzaState;

END_VAR
VAR
	Power : UINT;
	Init : BOOL;
	Timer : REAL;
	Timeout : REAL;
	TimerAspirazione : REAL;
	ParametersArray : ParametersArray;
	MAN_Actuator : UINT;
	MAN_Cmd : UINT;

	DistanzaFTC0 : REAL;
	DistanzaFTC180 : REAL;

	TimerPresaPiastrella : REAL;		
	DisattivazioneTotaleAspirazioni : bool;
	FiltroFTCFaldaSX : Signal_Filter;
	FiltroFTCFaldaDX : Signal_Filter;
	
	FTC_FaldaSXFiltrata : BOOL;
	FTC_FaldaDXFiltrata : bool;
	
	PostazionePrelievo : INT;
	
	AspiraSoloFalde : BOOL;//Se TRUE = si attiva solo l'aspirazione delle falde
	TempoRilascioInDeposito : REAL := 500;
END_VAR

IF NOT Init THEN
	TFCommandBufferClear(ADR(Cmd));
	TFCommandClear(ADR(CmdNext));
	TFCommandExeClear(ADR(CmdExe));
	TFStateUpdate(ADR(State),StateNOP);
	TFErrorClear(ADR(Error));
	TFWarningClear(ADR(Warning));
	Init := TRUE;
	CmdExe.Code := 1;
END_IF

(* Generic Timer - Add here all your Timers *)
TFTimerCall(ADR(Timer),Cfg.TimeBase);
TFTimerCall(ADR(Timeout),Cfg.TimeBase);
TFTimerCall(ADR(TimerPresaPiastrella),Cfg.TimeBase);
TFTimerCall(ADR(TimerAspirazione),Cfg.TimeBase);
(* External To Buffered Command *)
TFCommandToNext(ADR(Cmd),ADR(CmdNext),ADR(CmdExe),ADR(Cfg),ADR(Error),ADR(ErrorLog),ADR(State));

(* Buffered To Exe Command *)
TFCommandToExecution(ADR(CmdNext),ADR(CmdExe),ADR(Error),ADR(ErrorLog),ADR(State),ADR(CmdLog));

(* Chiamata FB *)
AspirazioneDX^();
AspirazioneSX^();
CilindroApertura^();
CilindroSbloccoRotazione^();
AspirazioneFaldaDX^();
AspirazioneFaldaSX^();

DistanzaFTC0 	:= Keyence_LRTB2000C(IN.InKeyence0_Byte0,IN.InKeyence0_Byte1);
DistanzaFTC180 	:= Keyence_LRTB2000C(IN.InKeyence180_Byte0,IN.InKeyence180_Byte1);

FiltroFTCFaldaDX(IN_Signal:=IN.FTC_FaldaDX,FilterTime_ON:=300,FilterTime_OFF:=300,Out_Signal_Filtrato=>FTC_FaldaDXFiltrata);
FiltroFTCFaldaSX(IN_Signal:=IN.FTC_FaldaSX,FilterTime_ON:=300,FilterTime_OFF:=300,Out_Signal_Filtrato=>FTC_FaldaSXFiltrata);


CASE Mission^.PPick OF
	
	1: PostazionePrelievo := RullP1;
	
	2: PostazionePrelievo := RullP2;

END_CASE


(* Exe Command *)
CASE CmdExe.Code OF

	(* ******************************************************************************************************** *)
	(* Nop  *)
	(* ******************************************************************************************************** *)
	CmdNOP:	;			
	(* ******************************************************************************************************** *)
	(* Stop *)
	(* ******************************************************************************************************** *)
	CmdSTOP:
		CASE CmdExe.CmdCase OF
			
			(* Case 0 *)
			0: 	TFStateUpdate(ADR(State),StateSTOP_RUN);
				TFTimerSet(ADR(Timeout),500,TRUE);
				TFCommandCase(ADR(CmdExe),1,CommandCase_INC);

			(* Case 1 - Clear All Commands*)
			1:	
				TFCommandCase(ADR(CmdExe),100,CommandCase_JMP);
			(* Case 100 *)
			100:TFStateUpdate(ADR(State),StateSTOP_END);
				TFCommandExeClear(ADR(CmdExe));

			ELSE
				TFError(ErrNOCMDCASE,ErrNULL,ADR(CmdExe),ADR(State),ADR(Error),ADR(ErrorLog));
		END_CASE;
	
	(* ******************************************************************************************************** *)
	(* Error Reset *)
	(* ******************************************************************************************************** *)
	CmdRESET:
		CASE CmdExe.CmdCase OF

			(* Case 0 *)
			0: 	TFStateUpdate(ADR(State),StateRESET_RUN);
				TFTimerSet(ADR(Timeout),2000+100,TRUE);
				TFTimerSet(ADR(Timer),2000,TRUE);
				TFCommandCase(ADR(CmdExe),1,CommandCase_INC);
			
			(* Case 1 - RESET COMANDI*)
			1: 
				TFClearAllCmdModulePinzaCompleta(AspirazioneDX,AspirazioneSX,CilindroApertura,CilindroSbloccoRotazione,AspirazioneFaldaDX,AspirazioneFaldaSX);
				TFCommandCase(ADR(CmdExe),1,CommandCase_INC);
			
			(* Case 2 - Invio comando di reset *)
			2:
				AspirazioneDX^.Command^.ErrorReset 				:= TRUE;	
				AspirazioneSX^.Command^.ErrorReset 				:= TRUE;	
				CilindroApertura^.Command.ErrorReset 			:= TRUE;	
				CilindroSbloccoRotazione^.Command.ErrorReset 	:= TRUE;	
				AspirazioneFaldaDX^.Command.ErrorReset 			:= TRUE;	
				AspirazioneFaldaSX^.Command.ErrorReset 			:= TRUE;	
				TFCommandCase(ADR(CmdExe),1,CommandCase_INC);
			
			(* Case 3 - Invio comando di reset *)
			3:
				IF AspirazioneDX^.Status.ErrorResetDone AND
					AspirazioneSX^.Status.ErrorResetDone AND
					CilindroApertura^.Status.ErrorResetDone AND
					CilindroSbloccoRotazione^.Status.ErrorResetDone AND
					AspirazioneFaldaDX^.Status.ErrorResetDone AND
					AspirazioneFaldaSX^.Status.ErrorResetDone THEN					
					TFClearAllCmdModulePinzaCompleta(AspirazioneDX,AspirazioneSX,CilindroApertura,CilindroSbloccoRotazione,AspirazioneFaldaDX,AspirazioneFaldaSX);
					TFCommandCase(ADR(CmdExe),99,CommandCase_JMP);
				ELSIF TFTimerDone(ADR(Timer)) THEN
					TFClearAllCmdModulePinzaCompleta(AspirazioneDX,AspirazioneSX,CilindroApertura,CilindroSbloccoRotazione,AspirazioneFaldaDX,AspirazioneFaldaSX);
					TFError(ErrTORESET,ErrNULL,ADR(CmdExe),ADR(State),ADR(Error),ADR(ErrorLog));
				END_IF

			(* Case 99 *)
			99:	TFErrorClear(ADR(Error));
				TFWarningClear(ADR(Warning));
				TFCommandCase(ADR(CmdExe),100,CommandCase_JMP);

			(* Case 100 *)
			100:TFStateUpdate(ADR(State),StateRESET_END);
				TFCommandExeClear(ADR(CmdExe));

			ELSE
				TFError(ErrNOCMDCASE,ErrNULL,ADR(CmdExe),ADR(State),ADR(Error),ADR(ErrorLog));
		END_CASE;

		(*IF AspirazioneDX^.Status.ErrorID <> ErrNULL THEN
			TFClearAllCmdModulePinza(AspirazioneDX,AspirazioneSX,CilindroApertura,CilindroSbloccoRotazione,AspirazioneFaldaDX,AspirazioneFaldaSX,CilindroTasteggio);
			TFError(ErrCYLINDER,AspirazioneDX^.Status.ErrorID,ADR(CmdExe),ADR(State),ADR(Error),ADR(ErrorLog));
		ELSIF AspirazioneSX^.Status.ErrorID <> ErrNULL THEN
			TFClearAllCmdModulePinza(AspirazioneDX,AspirazioneSX,CilindroApertura,CilindroSbloccoRotazione,AspirazioneFaldaDX,AspirazioneFaldaSX,CilindroTasteggio);
			TFError(ErrCYLINDER,AspirazioneSX^.Status.ErrorID,ADR(CmdExe),ADR(State),ADR(Error),ADR(ErrorLog));
		ELSIF CilindroApertura^.Status.ErrorID <> ErrNULL THEN
			TFClearAllCmdModulePinza(AspirazioneDX,AspirazioneSX,CilindroApertura,CilindroSbloccoRotazione,AspirazioneFaldaDX,AspirazioneFaldaSX,CilindroTasteggio);
			TFError(ErrCYLINDER,CilindroApertura^.Status.ErrorID,ADR(CmdExe),ADR(State),ADR(Error),ADR(ErrorLog));
		ELSIF CilindroSbloccoRotazione^.Status.ErrorID <> ErrNULL THEN
			TFClearAllCmdModulePinza(AspirazioneDX,AspirazioneSX,CilindroApertura,CilindroSbloccoRotazione,AspirazioneFaldaDX,AspirazioneFaldaSX,CilindroTasteggio);
			TFError(ErrCYLINDER,CilindroSbloccoRotazione^.Status.ErrorID,ADR(CmdExe),ADR(State),ADR(Error),ADR(ErrorLog));
		ELSIF AspirazioneFaldaDX^.Status.ErrorID <> ErrNULL THEN
			TFClearAllCmdModulePinza(AspirazioneDX,AspirazioneSX,CilindroApertura,CilindroSbloccoRotazione,AspirazioneFaldaDX,AspirazioneFaldaSX,CilindroTasteggio);
			TFError(ErrCYLINDER,AspirazioneFaldaDX^.Status.ErrorID,ADR(CmdExe),ADR(State),ADR(Error),ADR(ErrorLog));
		ELSIF AspirazioneFaldaSX^.Status.ErrorID <> ErrNULL THEN
			TFClearAllCmdModulePinza(AspirazioneDX,AspirazioneSX,CilindroApertura,CilindroSbloccoRotazione,AspirazioneFaldaDX,AspirazioneFaldaSX,CilindroTasteggio);
			TFError(ErrCYLINDER,AspirazioneFaldaSX^.Status.ErrorID,ADR(CmdExe),ADR(State),ADR(Error),ADR(ErrorLog));
		*)
		IF TFTimerDone(ADR(Timeout)) THEN
			TFClearAllCmdModulePinzaCompleta(AspirazioneDX,AspirazioneSX,CilindroApertura,CilindroSbloccoRotazione,AspirazioneFaldaDX,AspirazioneFaldaSX);
			TFError(ErrCMDTIMEOUT,ErrNULL,ADR(CmdExe),ADR(State),ADR(Error),ADR(ErrorLog));
		END_IF
	
	(* ******************************************************************************************************** *)
	(* Power *)
	(* ******************************************************************************************************** *)
	CmdPOWER:
		CASE CmdExe.CmdCase OF
			
			(* Case 0 *)
			0: 	TFStateUpdate(ADR(State),StatePOWER_RUN);
				TFTimerSet(ADR(Timeout),500,TRUE);
				TFCommandCase(ADR(CmdExe),100,CommandCase_JMP);

			1: TFCommandCase(ADR(CmdExe),100,CommandCase_JMP);
			(* Case 100 *)
			100:TFStateUpdate(ADR(State),StatePOWER_END);
				TFCommandExeClear(ADR(CmdExe));

			ELSE
				TFError(ErrNOCMDCASE,ErrNULL,ADR(CmdExe),ADR(State),ADR(Error),ADR(ErrorLog));
		END_CASE
	
	(* ******************************************************************************************************** *)
	(* Home *)
	(* ******************************************************************************************************** *)
	CmdHOME:
		CASE CmdExe.CmdCase OF

			(* Case 0 *)
			0: 	TFStateUpdate(ADR(State),StateHOME_RUN);
				TFTimerSet(ADR(Timeout),3000+200,TRUE);
				TFTimerSet(ADR(Timer),3000,TRUE);
				TFCommandCase(ADR(CmdExe),1,CommandCase_INC);

			(* Case 1 - *)
			1: 
				TFCommandCase(ADR(CmdExe),10,CommandCase_JMP);

			(* Case 10 - Set automatico Soglie *)
			10:
				AspirazioneDX^.Command^.Aspirazione_ON_ScritturaSoglia 	:= TRUE;
				AspirazioneSX^.Command^.Aspirazione_ON_ScritturaSoglia 	:= TRUE;
				IF AspirazioneDX^.Status.CommandDone AND AspirazioneSX^.Status.CommandDone THEN
					AspirazioneDX^.Command^.Aspirazione_ON_ScritturaSoglia		:= FALSE;
					AspirazioneSX^.Command^.Aspirazione_ON_ScritturaSoglia		:= FALSE;
					TFCommandCase(ADR(CmdExe),100,CommandCase_JMP);
				ELSIF TFTimerDone(ADR(Timer)) THEN
					AspirazioneDX^.Command^.Aspirazione_ON_ScritturaSoglia		:= FALSE;
					AspirazioneSX^.Command^.Aspirazione_ON_ScritturaSoglia		:= FALSE;
					TFError(ErrTOHOME,ErrNULL,ADR(CmdExe),ADR(State),ADR(Error),ADR(ErrorLog));
				END_IF
			
	
			(* Case 100 *)
			100:TFStateUpdate(ADR(State),StateHOME_END);
				TFCommandExeClear(ADR(CmdExe));

			ELSE
				TFError(ErrNOCMDCASE,ErrNULL,ADR(CmdExe),ADR(State),ADR(Error),ADR(ErrorLog));
		END_CASE;
		
		IF AspirazioneDX^.Status.ErrorID <> ErrNULL THEN
			AspirazioneDX^.Command^.Aspirazione_ON_ScritturaSoglia 	:= TRUE;
			AspirazioneSX^.Command^.Aspirazione_ON_ScritturaSoglia 	:= TRUE;
			TFError(ErrCYLINDER,AspirazioneDX^.Status.ErrorID,ADR(CmdExe),ADR(State),ADR(Error),ADR(ErrorLog));
		ELSIF AspirazioneSX^.Status.ErrorID <> ErrNULL THEN
			AspirazioneDX^.Command^.Aspirazione_ON_ScritturaSoglia 	:= TRUE;
			AspirazioneSX^.Command^.Aspirazione_ON_ScritturaSoglia 	:= TRUE;
			TFError(ErrCYLINDER,AspirazioneSX^.Status.ErrorID,ADR(CmdExe),ADR(State),ADR(Error),ADR(ErrorLog));
		ELSIF CilindroApertura^.Status.ErrorID <> ErrNULL THEN
			AspirazioneDX^.Command^.Aspirazione_ON_ScritturaSoglia 	:= TRUE;
			AspirazioneSX^.Command^.Aspirazione_ON_ScritturaSoglia 	:= TRUE;
			TFError(ErrCYLINDER,CilindroApertura^.Status.ErrorID,ADR(CmdExe),ADR(State),ADR(Error),ADR(ErrorLog));
		ELSIF CilindroSbloccoRotazione^.Status.ErrorID <> ErrNULL THEN
			AspirazioneDX^.Command^.Aspirazione_ON_ScritturaSoglia 	:= TRUE;
			AspirazioneSX^.Command^.Aspirazione_ON_ScritturaSoglia 	:= TRUE;
			TFError(ErrCYLINDER,CilindroSbloccoRotazione^.Status.ErrorID,ADR(CmdExe),ADR(State),ADR(Error),ADR(ErrorLog));
		ELSIF AspirazioneFaldaDX^.Status.ErrorID <> ErrNULL THEN
			AspirazioneDX^.Command^.Aspirazione_ON_ScritturaSoglia 	:= TRUE;
			AspirazioneSX^.Command^.Aspirazione_ON_ScritturaSoglia 	:= TRUE;
			TFError(ErrCYLINDER,AspirazioneFaldaDX^.Status.ErrorID,ADR(CmdExe),ADR(State),ADR(Error),ADR(ErrorLog));
		ELSIF AspirazioneFaldaSX^.Status.ErrorID <> ErrNULL THEN
			AspirazioneDX^.Command^.Aspirazione_ON_ScritturaSoglia 	:= TRUE;
			AspirazioneSX^.Command^.Aspirazione_ON_ScritturaSoglia 	:= TRUE;
			TFError(ErrCYLINDER,AspirazioneFaldaSX^.Status.ErrorID,ADR(CmdExe),ADR(State),ADR(Error),ADR(ErrorLog));
		ELSIF TFTimerDone(ADR(Timeout)) THEN
			AspirazioneDX^.Command^.Aspirazione_ON_ScritturaSoglia 	:= TRUE;
			AspirazioneSX^.Command^.Aspirazione_ON_ScritturaSoglia 	:= TRUE;
			TFError(ErrCMDTIMEOUT,ErrNULL,ADR(CmdExe),ADR(State),ADR(Error),ADR(ErrorLog));
		END_IF

	(* ******************************************************************************************************** *)
	(* Manual *)
	(* ******************************************************************************************************** *)
	CmdMAN:
		CASE CmdExe.CmdCase OF
			(* Case 0 *)
			0: 	TFStateUpdate(ADR(State),StateMAN_RUN);
				TFTimerSet(ADR(Timeout),3000,TRUE);
				IF TFCommandParRead(CmdExe.Cmd.Parameter,ADR(ParametersArray),2) THEN
					MAN_Actuator	:= STRING_TO_UINT(ParametersArray.Parameters[0]);
					MAN_Cmd		:= STRING_TO_UINT(ParametersArray.Parameters[1]);
				ELSE
					TFError(ErrCMDPARNUM,ErrNULL,ADR(CmdExe),ADR(State),ADR(Error),ADR(ErrorLog));
					RETURN;
				END_IF;

				CASE MAN_Actuator OF
					(* Case 0..99 for Actuators *)
					(* Case 100..199  for Axis *)

					(* Case Nop *)
					0:	;

					(* Case 1: *)
					1:	CASE MAN_Cmd OF
							0:	;
							
							(* Case 10: Apertura Pinza *)
							10:	
								CilindroApertura^.Command.Activation 	:= TRUE;
								CilindroApertura^.Command.Deactivation 	:= FALSE;
								TFTimerSet(ADR(Timeout),30000,TRUE);
								TFCommandCase(ADR(CmdExe),10,CommandCase_JMP);
								
							(* Case 11: Chiusura Pinza *)
							11:	
								CilindroApertura^.Command.Activation 	:= FALSE;
								CilindroApertura^.Command.Deactivation 	:= TRUE;
								TFTimerSet(ADR(Timeout),30000,TRUE);
								TFCommandCase(ADR(CmdExe),10,CommandCase_JMP);

							(* Case 20: Sgancio Sblocco Rotazione *)
							20:	
								CilindroSbloccoRotazione^.Command.Activation 	:= TRUE;
								CilindroSbloccoRotazione^.Command.Deactivation 	:= FALSE;
								TFTimerSet(ADR(Timeout),3000,TRUE);
								TFCommandCase(ADR(CmdExe),20,CommandCase_JMP);
								
							(* Case 21: Aggancio Sblocco Rotazione *)
							21:	
								CilindroSbloccoRotazione^.Command.Activation 	:= FALSE;
								CilindroSbloccoRotazione^.Command.Deactivation 	:= TRUE;
								TFTimerSet(ADR(Timeout),3000,TRUE);
								TFCommandCase(ADR(CmdExe),20,CommandCase_JMP);

							(* Case 30: Ativazione Aspirazione Falda DX *)
							30:	
								AspirazioneFaldaDX^.Command.Activation 		:= TRUE;
								AspirazioneFaldaDX^.Command.Deactivation 	:= FALSE;
								TFTimerSet(ADR(Timeout),3000,TRUE);
								TFCommandCase(ADR(CmdExe),30,CommandCase_JMP);
								
							(* Case 31: Disattivazione Aspirazione Falda DX *)
							31:	
								AspirazioneFaldaDX^.Command.Activation 		:= FALSE;
								AspirazioneFaldaDX^.Command.Deactivation 	:= TRUE;
								TFTimerSet(ADR(Timeout),3000,TRUE);
								TFCommandCase(ADR(CmdExe),30,CommandCase_JMP);
								
							(* Case 40: Ativazione Aspirazione Falda SX *)
							40:	
								AspirazioneFaldaSX^.Command.Activation 		:= TRUE;
								AspirazioneFaldaSX^.Command.Deactivation 	:= FALSE;

								TFTimerSet(ADR(Timeout),3000,TRUE);
								TFCommandCase(ADR(CmdExe),40,CommandCase_JMP);
								
							(* Case 41: Disattivazione Aspirazione Falda SX *)
							41:	
								AspirazioneFaldaSX^.Command.Activation 		:= FALSE;
								AspirazioneFaldaSX^.Command.Deactivation 	:= TRUE;

								TFTimerSet(ADR(Timeout),3000,TRUE);
								TFCommandCase(ADR(CmdExe),40,CommandCase_JMP);

							(* Case 50: Ativazione Aspirazione SX *)
							50:	
								AspirazioneSX^.Command^.Aspirazione_ON 	:= TRUE;
								AspirazioneSX^.Command^.Aspirazione_OFF := FALSE;

								AspirazioneDX^.Command^.Aspirazione_ON 	:= TRUE;
								AspirazioneDX^.Command^.Aspirazione_OFF := FALSE;

								TFTimerSet(ADR(Timeout),3000,TRUE);
								TFCommandCase(ADR(CmdExe),50,CommandCase_JMP);
								
							(* Case 51: Disattivazione Aspirazione SX *)
							51:	
								AspirazioneSX^.Command^.Aspirazione_ON 	:= FALSE;
								AspirazioneSX^.Command^.Aspirazione_OFF := TRUE;
								TFTimerSet(ADR(Timeout),3000,TRUE);
								TFCommandCase(ADR(CmdExe),50,CommandCase_JMP);

							(* Case 60: Ativazione Aspirazione DX *)
							60:	
								AspirazioneDX^.Command^.Aspirazione_ON 	:= TRUE;
								AspirazioneDX^.Command^.Aspirazione_OFF := FALSE;
								TFTimerSet(ADR(Timeout),3000,TRUE);
								TFCommandCase(ADR(CmdExe),60,CommandCase_JMP);
								
							(* Case 61: Disattivazione Aspirazione SX *)
							61:	
								AspirazioneDX^.Command^.Aspirazione_ON 	:= FALSE;
								AspirazioneDX^.Command^.Aspirazione_OFF := TRUE;
								AspirazioneSX^.Command^.Aspirazione_ON 	:= FALSE;
								AspirazioneSX^.Command^.Aspirazione_OFF := TRUE;
								StatoPinza.ElementoPrelevato := FALSE;
								TFTimerSet(ADR(Timeout),3000,TRUE);
								TFCommandCase(ADR(CmdExe),60,CommandCase_JMP);
				
							(* Case 70: Ativazione Tastatori *)
							70:	
								//CilindroTasteggio^.Command.Activation 		:= TRUE;
								//CilindroTasteggio^.Command.Deactivation 	:= FALSE;
								TFTimerSet(ADR(Timeout),3000,TRUE);
								TFCommandCase(ADR(CmdExe),70,CommandCase_JMP);
								
							(* Case 71: Disattivazione Aspirazione SX *)
							71:	
								//CilindroTasteggio^.Command.Activation 		:= FALSE;
								//CilindroTasteggio^.Command.Deactivation 	:= TRUE;
								TFTimerSet(ADR(Timeout),3000,TRUE);
								TFCommandCase(ADR(CmdExe),70,CommandCase_JMP);

							ELSE
								TFError(ErrNOCMDCASE,ErrNULL,ADR(CmdExe),ADR(State),ADR(Error),ADR(ErrorLog));
						END_CASE;

					100:CASE MAN_Cmd OF
							0:	;
							ELSE
								TFError(ErrNOCMDCASE,ErrNULL,ADR(CmdExe),ADR(State),ADR(Error),ADR(ErrorLog));
						END_CASE;

					ELSE
						TFError(ErrNOCMDCASE,ErrNULL,ADR(CmdExe),ADR(State),ADR(Error),ADR(ErrorLog));
				END_CASE;

				//IF CmdExe.CmdCase = 0 THEN
					//TFCommandCase(ADR(CmdExe),1,CommandCase_INC);
				//END_IF

			(* Case 1 - *)
			1: 	IF (MAN_Cmd = 0) OR TFTimerDone(ADR(Timeout)) THEN
					(* Clear All Output Here *)
					;
					TFStateUpdate(ADR(State),StateMAN_END);
					TFCommandExeClear(ADR(CmdExe));
				END_IF;

			
			(* Case 10 - CilindroApertura *)
			10: 
				IF CilindroApertura^.Status.CommandDone THEN
					CilindroApertura^.Command.Activation 	:= FALSE;
					CilindroApertura^.Command.Deactivation 	:= FALSE;
					TFCommandCase(ADR(CmdExe),100,CommandCase_JMP);
				ELSIF CilindroApertura^.Status.ErrorID <> ErrNULL THEN
					TFClearAllCmdModulePinzaCompleta(AspirazioneDX,AspirazioneSX,CilindroApertura,CilindroSbloccoRotazione,AspirazioneFaldaDX,AspirazioneFaldaSX);
					TFError(ErrCYLINDER,CilindroApertura^.Status.ErrorID,ADR(CmdExe),ADR(State),ADR(Error),ADR(ErrorLog));
				END_IF

			(* Case 20 - CilindroSbloccoRotazione *)
			20: 
				IF CilindroSbloccoRotazione^.Status.CommandDone THEN
					CilindroSbloccoRotazione^.Command.Activation 	:= FALSE;
					CilindroSbloccoRotazione^.Command.Deactivation 	:= FALSE;
					TFCommandCase(ADR(CmdExe),100,CommandCase_JMP);
				ELSIF CilindroSbloccoRotazione^.Status.ErrorID <> ErrNULL THEN
					TFClearAllCmdModulePinzaCompleta(AspirazioneDX,AspirazioneSX,CilindroApertura,CilindroSbloccoRotazione,AspirazioneFaldaDX,AspirazioneFaldaSX);
					TFError(ErrCYLINDER,CilindroSbloccoRotazione^.Status.ErrorID,ADR(CmdExe),ADR(State),ADR(Error),ADR(ErrorLog));
				END_IF

			(* Case 30 - AspirazioneFaldaDX *)
			30: 
				IF AspirazioneFaldaDX^.Status.CommandDone THEN
					AspirazioneFaldaDX^.Command.Activation 	:= FALSE;
					AspirazioneFaldaDX^.Command.Deactivation 	:= FALSE;
					TFCommandCase(ADR(CmdExe),100,CommandCase_JMP);
				ELSIF AspirazioneFaldaDX^.Status.ErrorID <> ErrNULL THEN
					TFClearAllCmdModulePinzaCompleta(AspirazioneDX,AspirazioneSX,CilindroApertura,CilindroSbloccoRotazione,AspirazioneFaldaDX,AspirazioneFaldaSX);
					TFError(ErrCYLINDER,AspirazioneFaldaDX^.Status.ErrorID,ADR(CmdExe),ADR(State),ADR(Error),ADR(ErrorLog));
				END_IF

			(* Case 40 - AspirazioneFaldaSX *)
			40: 
				IF AspirazioneFaldaSX^.Status.CommandDone THEN
					AspirazioneFaldaSX^.Command.Activation 	:= FALSE;
					AspirazioneFaldaSX^.Command.Deactivation 	:= FALSE;
					TFCommandCase(ADR(CmdExe),100,CommandCase_JMP);
				ELSIF AspirazioneFaldaSX^.Status.ErrorID <> ErrNULL THEN
					TFClearAllCmdModulePinzaCompleta(AspirazioneDX,AspirazioneSX,CilindroApertura,CilindroSbloccoRotazione,AspirazioneFaldaDX,AspirazioneFaldaSX);
					TFError(ErrCYLINDER,AspirazioneFaldaSX^.Status.ErrorID,ADR(CmdExe),ADR(State),ADR(Error),ADR(ErrorLog));
				END_IF

			(* Case 50 - AspirazioneSX *)
			50: 
				IF AspirazioneSX^.Status.CommandDone AND AspirazioneDX^.Status.CommandDone THEN
					AspirazioneDX^.Command^.Aspirazione_ON 	:= FALSE;
					AspirazioneDX^.Command^.Aspirazione_OFF	:= FALSE;
					AspirazioneSX^.Command^.Aspirazione_ON 	:= FALSE;
					AspirazioneSX^.Command^.Aspirazione_OFF	:= FALSE;
					TFCommandCase(ADR(CmdExe),100,CommandCase_JMP);
				ELSIF AspirazioneSX^.Status.ErrorID <> ErrNULL THEN
					TFClearAllCmdModulePinzaCompleta(AspirazioneDX,AspirazioneSX,CilindroApertura,CilindroSbloccoRotazione,AspirazioneFaldaDX,AspirazioneFaldaSX);
					TFError(ErrCYLINDER,AspirazioneSX^.Status.ErrorID,ADR(CmdExe),ADR(State),ADR(Error),ADR(ErrorLog));
				ELSIF AspirazioneDX^.Status.ErrorID <> ErrNULL THEN
					TFClearAllCmdModulePinzaCompleta(AspirazioneDX,AspirazioneSX,CilindroApertura,CilindroSbloccoRotazione,AspirazioneFaldaDX,AspirazioneFaldaSX);
					TFError(ErrCYLINDER,AspirazioneDX^.Status.ErrorID,ADR(CmdExe),ADR(State),ADR(Error),ADR(ErrorLog));
				END_IF

